C05355=1014.122,185.886,-129.232,167.084,55.090,160.182
C05356=1014.126,186.134,-129.253,167.087,55.079,160.180
C05357=1014.130,186.414,-129.276,167.092,55.066,160.179
C05358=1014.134,186.693,-129.300,167.097,55.052,160.177
C05359=1014.140,186.972,-129.324,167.102,55.039,160.176
C05360=1014.144,187.252,-129.348,167.107,55.025,160.174
C05361=1014.148,187.500,-129.369,167.111,55.014,160.173
C05362=1014.152,187.750,-129.391,167.116,55.002,160.171
C05363=1014.156,187.999,-129.411,167.120,54.990,160.170
C05364=1014.160,188.248,-129.433,167.124,54.979,160.168
C05365=1014.164,188.496,-129.454,167.129,54.967,160.167
C05366=1014.168,188.746,-129.476,167.134,54.955,160.166
C05367=1014.172,188.995,-129.497,167.137,54.943,160.164
C05368=1014.177,189.244,-129.518,167.142,54.931,160.163
C05369=1014.180,189.493,-129.538,167.146,54.920,160.161
C05370=1014.184,189.743,-129.560,167.150,54.908,160.160
C05371=1014.188,189.991,-129.582,167.155,54.896,160.159
C05372=1014.193,190.240,-129.603,167.160,54.885,160.157
C05373=1014.197,190.490,-129.624,167.164,54.873,160.156
C05374=1014.201,190.739,-129.645,167.168,54.861,160.154
C05375=1014.205,190.988,-129.667,167.172,54.849,160.153
C05376=1014.209,191.236,-129.688,167.177,54.837,160.151
C05377=1014.213,191.486,-129.710,167.181,54.826,160.150
C05378=1014.217,191.734,-129.731,167.186,54.814,160.149
C05379=1014.222,191.984,-129.752,167.190,54.802,160.147
C05380=1014.226,192.233,-129.774,167.195,54.790,160.146
C05381=1014.230,192.482,-129.795,167.199,54.778,160.144
C05382=1014.234,192.731,-129.817,167.203,54.767,160.143
C05383=1014.238,192.980,-129.838,167.208,54.755,160.142
C05384=1014.243,193.228,-129.859,167.213,54.743,160.140
C05385=1014.247,193.478,-129.881,167.218,54.731,160.139
C05386=1014.251,193.727,-129.902,167.222,54.719,160.137
C05387=1014.256,193.976,-129.924,167.226,54.707,160.136
C05388=1014.259,194.225,-129.946,167.231,54.696,160.135
C05389=1014.263,194.474,-129.966,167.235,54.684,160.133
C05390=1014.268,194.723,-129.988,167.240,54.672,160.132
C05391=1014.273,194.972,-130.009,167.245,54.660,160.131
C05392=1014.276,195.221,-130.031,167.249,54.648,160.129
C05393=1014.281,195.470,-130.053,167.253,54.637,160.127
C05394=1014.286,195.719,-130.074,167.258,54.625,160.126
C05395=1014.289,195.969,-130.096,167.263,54.613,160.125
C05396=1014.293,196.218,-130.117,167.267,54.601,160.123
C05397=1014.298,196.466,-130.139,167.272,54.589,160.122
C05398=1014.303,196.716,-130.160,167.277,54.577,160.121
C05399=1014.306,196.964,-130.182,167.282,54.565,160.119
C05400=1014.311,197.214,-130.203,167.287,54.554,160.118
C05401=1014.315,197.462,-130.225,167.290,54.542,160.116
C05402=1014.320,197.712,-130.246,167.295,54.530,160.115
C05403=1014.323,197.960,-130.268,167.300,54.518,160.114
C05404=1014.328,198.209,-130.290,167.304,54.507,160.112
C05405=1014.333,198.459,-130.311,167.309,54.495,160.111
C05406=1014.337,198.708,-130.334,167.314,54.482,160.109
C05407=1014.341,198.957,-130.355,167.319,54.471,160.108
C05408=1014.345,199.206,-130.377,167.323,54.459,160.107
C05409=1014.350,199.454,-130.399,167.328,54.447,160.105
C05410=1014.354,199.704,-130.421,167.333,54.436,160.104
C05411=1014.358,199.953,-130.443,167.337,54.424,160.103
C05412=1014.362,200.202,-130.465,167.342,54.413,160.101
C05413=1014.366,200.451,-130.487,167.347,54.401,160.100
C05414=1014.370,200.700,-130.510,167.352,54.389,160.099
C05415=1014.375,200.948,-130.531,167.357,54.378,160.097
C05416=1014.379,201.198,-130.554,167.362,54.366,160.096
C05417=1014.383,201.447,-130.576,167.366,54.354,160.095
C05418=1014.387,201.696,-130.597,167.371,54.342,160.093
C05419=1014.391,201.945,-130.620,167.375,54.331,160.092
C05420=1014.395,202.194,-130.642,167.380,54.319,160.090
C05421=1014.415,203.311,-130.741,167.905,54.401,160.226
C05422=1014.420,203.543,-130.764,167.909,54.392,160.225
C05423=1014.424,203.777,-130.786,167.913,54.381,160.223
C05424=1014.429,204.010,-130.808,167.918,54.371,160.222
C05425=1014.435,204.242,-130.831,167.921,54.361,160.221
C05426=1014.439,204.475,-130.853,167.926,54.351,160.220
C05427=1014.444,204.708,-130.875,167.930,54.341,160.218
C05428=1014.449,204.940,-130.897,167.934,54.331,160.217
C05429=1014.454,205.173,-130.919,167.939,54.322,160.216
C05430=1014.460,205.422,-130.944,167.943,54.311,160.215
C05431=1014.465,205.671,-130.967,167.947,54.301,160.213
C05432=1014.470,205.920,-130.991,167.952,54.290,160.212
C05433=1014.475,206.168,-131.016,167.956,54.280,160.211
C05434=1014.481,206.418,-131.040,167.960,54.269,160.210
C05435=1014.486,206.667,-131.064,167.964,54.258,160.208
C05436=1014.491,206.915,-131.088,167.969,54.248,160.207
C05437=1014.497,207.164,-131.112,167.974,54.237,160.206
C05438=1014.502,207.413,-131.137,167.978,54.227,160.204
C05439=1014.507,207.662,-131.160,167.983,54.217,160.203
C05440=1014.512,207.910,-131.184,167.987,54.206,160.202
C05441=1014.518,208.159,-131.209,167.992,54.196,160.201
C05442=1014.523,208.408,-131.233,167.996,54.185,160.199
C05443=1014.528,208.656,-131.257,168.000,54.175,160.198
C05444=1014.533,208.905,-131.281,168.005,54.165,160.197
C05445=1014.538,209.154,-131.305,168.009,54.154,160.196
C05446=1014.544,209.403,-131.329,168.014,54.144,160.194
C05447=1014.550,209.652,-131.354,168.019,54.134,160.193
C05448=1014.554,209.901,-131.379,168.023,54.124,160.192
C05449=1014.559,210.149,-131.403,168.027,54.113,160.191
C05450=1014.565,210.398,-131.427,168.032,54.103,160.190
C05451=1014.570,210.646,-131.452,168.036,54.093,160.188
C05452=1014.575,210.895,-131.476,168.040,54.083,160.187
C05453=1014.580,211.144,-131.501,168.044,54.073,160.186
C05454=1014.586,211.393,-131.525,168.049,54.063,160.185
C05455=1014.591,211.642,-131.550,168.054,54.053,160.184
C05456=1014.596,211.890,-131.574,168.058,54.042,160.182
C05457=1014.601,212.139,-131.599,168.063,54.032,160.181
C05458=1014.606,212.388,-131.623,168.067,54.022,160.180
C05459=1014.613,212.637,-131.648,168.072,54.012,160.179
C05460=1014.618,212.885,-131.672,168.076,54.002,160.178
C05461=1014.622,213.134,-131.697,168.081,53.992,160.176
C05462=1014.628,213.383,-131.722,168.084,53.982,160.175
C05463=1014.633,213.631,-131.746,168.089,53.972,160.174
C05464=1014.639,213.881,-131.770,168.094,53.962,160.173
C05465=1014.644,214.129,-131.795,168.098,53.952,160.172
C05466=1014.649,214.378,-131.820,168.103,53.942,160.171
C05467=1014.654,214.626,-131.845,168.108,53.932,160.169
C05468=1014.660,214.875,-131.869,168.113,53.922,160.168
C05469=1014.666,215.124,-131.893,168.116,53.913,160.167
C05470=1014.670,215.373,-131.918,168.121,53.902,160.166
C05471=1014.676,215.622,-131.943,168.126,53.892,160.165
C05472=1014.682,215.870,-131.968,168.130,53.883,160.164
C05473=1014.687,216.119,-131.992,168.135,53.872,160.162
C05474=1014.691,216.367,-132.017,168.140,53.863,160.161
C05475=1014.697,216.617,-132.042,168.144,53.853,160.160
C05476=1014.703,216.865,-132.067,168.148,53.843,160.159
C05477=1014.708,217.113,-132.091,168.153,53.833,160.158
C05478=1014.714,217.363,-132.115,168.158,53.823,160.157
C05479=1014.719,217.612,-132.140,168.163,53.814,160.156
C05480=1014.724,217.859,-132.165,168.166,53.803,160.154
C05481=1014.730,218.108,-132.190,168.171,53.794,160.153
C05482=1014.735,218.355,-132.215,168.176,53.784,160.152
C05483=1014.740,218.600,-132.239,168.179,53.775,160.151
C05484=1014.745,218.846,-132.264,168.184,53.765,160.150
C05485=1014.750,219.092,-132.289,168.188,53.756,160.149
C05486=1014.756,219.338,-132.314,168.193,53.746,160.147
C05487=1014.761,219.584,-132.340,168.197,53.737,160.147
C05488=1014.766,219.829,-132.364,168.202,53.728,160.145
C05489=1014.771,220.075,-132.389,168.206,53.718,160.144
C05490=1014.777,220.324,-132.413,168.211,53.709,160.143
C05491=1014.782,220.573,-132.439,168.216,53.699,160.142
C05492=1014.787,220.821,-132.463,168.220,53.690,160.141
C05493=1014.793,221.070,-132.489,168.225,53.680,160.140
C05494=1014.798,221.318,-132.514,168.230,53.670,160.139
C05495=1014.803,221.568,-132.539,168.234,53.661,160.138
C05496=1014.809,221.816,-132.564,168.238,53.651,160.137
C05497=1014.814,222.065,-132.590,168.243,53.641,160.136
C05498=1014.820,222.313,-132.615,168.247,53.632,160.134
C05499=1014.825,222.562,-132.640,168.252,53.622,160.133
C05500=1014.831,222.811,-132.665,168.257,53.614,160.132
C05501=1014.835,223.059,-132.690,168.261,53.604,160.131
C05502=1014.842,223.308,-132.716,168.266,53.594,160.130
C05503=1014.846,223.557,-132.740,168.270,53.585,160.129
C05504=1014.852,223.806,-132.766,168.275,53.575,160.128
C05505=1014.857,224.054,-132.791,168.279,53.566,160.127
C05506=1014.862,224.303,-132.817,168.285,53.557,160.126
C05507=1014.868,224.551,-132.842,168.288,53.548,160.125
C05508=1014.873,224.800,-132.868,168.293,53.538,160.124
C05509=1014.880,225.049,-132.893,168.298,53.528,160.123
C05510=1014.884,225.298,-132.918,168.303,53.520,160.122
C05511=1014.890,225.547,-132.943,168.308,53.510,160.121
C05512=1014.895,225.795,-132.969,168.312,53.501,160.120
C05513=1014.902,226.044,-132.994,168.317,53.492,160.119
C05514=1014.906,226.292,-133.020,168.321,53.483,160.118
C05515=1014.912,226.541,-133.045,168.326,53.473,160.117
C05516=1014.916,226.790,-133.070,168.330,53.464,160.116
C05517=1014.922,227.039,-133.096,168.335,53.455,160.115
C05518=1014.928,227.287,-133.122,168.340,53.446,160.114
C05519=1014.933,227.536,-133.147,168.343,53.437,160.112
C05520=1014.938,227.785,-133.173,168.349,53.428,160.112
C05521=1014.943,228.033,-133.199,168.353,53.419,160.110
C05522=1014.949,228.282,-133.224,168.358,53.410,160.110
C05523=1014.955,228.531,-133.250,168.362,53.400,160.108
C05524=1014.960,228.779,-133.275,168.368,53.392,160.108
C05525=1014.965,229.028,-133.301,168.372,53.382,160.106
C05526=1014.970,229.276,-133.327,168.376,53.374,160.105
C05527=1014.977,229.524,-133.353,168.381,53.365,160.105
C05528=1014.982,229.773,-133.379,168.385,53.355,160.103
C05529=1014.987,230.021,-133.405,168.391,53.347,160.103
C05530=1014.992,230.270,-133.430,168.395,53.338,160.102
C05531=1014.998,230.519,-133.456,168.399,53.329,160.101
C05532=1015.003,230.768,-133.482,168.405,53.320,160.100
C05533=1015.009,231.016,-133.509,168.409,53.311,160.099
C05534=1015.014,231.265,-133.535,168.413,53.303,160.098
C05535=1015.019,231.513,-133.560,168.418,53.293,160.097
C05536=1015.024,231.762,-133.586,168.423,53.284,160.096
C05537=1015.030,232.011,-133.612,168.427,53.276,160.095
C05538=1015.035,232.259,-133.638,168.432,53.267,160.094
C05539=1015.040,232.508,-133.664,168.437,53.258,160.093
C05540=1015.046,232.757,-133.690,168.441,53.249,160.092
C05541=1015.051,233.004,-133.716,168.445,53.241,160.091
C05542=1015.057,233.246,-133.742,168.450,53.232,160.090
C05543=1015.062,233.488,-133.767,168.454,53.224,160.089
C05544=1015.068,233.730,-133.792,168.460,53.215,160.088
C05545=1015.072,233.972,-133.818,168.465,53.207,160.088
C05546=1015.078,234.213,-133.843,168.469,53.198,160.087
C05547=1015.083,234.455,-133.868,168.474,53.190,160.086
C05548=1015.089,234.697,-133.893,168.478,53.181,160.085
C05549=1015.094,234.938,-133.918,168.483,53.173,160.084
C05550=1015.100,235.187,-133.945,168.487,53.164,160.083
C05551=1015.105,235.436,-133.971,168.491,53.156,160.082
C05552=1015.111,235.684,-133.997,168.497,53.147,160.081
C05553=1015.116,235.933,-134.023,168.501,53.138,160.080
C05554=1015.121,236.181,-134.049,168.506,53.130,160.079
C05555=1015.127,236.430,-134.075,168.510,53.121,160.078
C05556=1015.132,236.679,-134.101,168.515,53.113,160.077
C05557=1015.138,236.927,-134.128,168.520,53.104,160.076
C05558=1015.144,237.176,-134.154,168.525,53.095,160.076
C05559=1015.149,237.424,-134.181,168.530,53.087,160.075
C05560=1015.154,237.673,-134.206,168.534,53.079,160.074
C05561=1015.159,237.921,-134.233,168.538,53.070,160.073
C05562=1015.165,238.170,-134.260,168.544,53.061,160.072
C05563=1015.171,238.419,-134.286,168.548,53.053,160.071
C05564=1015.176,238.667,-134.313,168.553,53.044,160.070
C05565=1015.182,238.915,-134.339,168.558,53.037,160.070
C05566=1015.187,239.164,-134.365,168.562,53.028,160.069
C05567=1015.193,239.412,-134.392,168.567,53.020,160.068
C05568=1015.198,239.661,-134.419,168.572,53.012,160.067
C05569=1015.204,239.909,-134.445,168.576,53.003,160.066
C05570=1015.209,240.158,-134.471,168.582,52.994,160.065
C05571=1015.214,240.407,-134.499,168.587,52.987,160.064
C05572=1015.220,240.655,-134.525,168.591,52.978,160.064
C05573=1015.226,240.903,-134.552,168.596,52.970,160.063
C05574=1015.230,241.153,-134.578,168.600,52.962,160.062
C05575=1015.236,241.401,-134.605,168.605,52.953,160.061
C05576=1015.242,241.649,-134.632,168.610,52.946,160.060
C05577=1015.248,241.898,-134.658,168.614,52.937,160.059
C05578=1015.253,242.146,-134.686,168.619,52.929,160.059
C05579=1015.258,242.394,-134.712,168.624,52.921,160.058
C05580=1015.264,242.642,-134.739,168.629,52.913,160.057
C05581=1015.269,242.891,-134.766,168.633,52.905,160.056
C05582=1015.275,243.139,-134.792,168.638,52.897,160.055
C05583=1015.280,243.388,-134.820,168.643,52.888,160.054
C05584=1015.285,243.636,-134.846,168.648,52.880,160.054
C05585=1015.290,243.885,-134.874,168.653,52.873,160.053
C05586=1015.295,244.134,-134.901,168.657,52.864,160.052
C05587=1015.301,244.382,-134.927,168.662,52.856,160.051
C05588=1015.306,244.631,-134.955,168.667,52.849,160.051
C05589=1015.312,244.879,-134.981,168.672,52.841,160.050
C05590=1015.317,245.127,-135.009,168.676,52.832,160.049
C05591=1015.322,245.376,-135.037,168.681,52.825,160.048
C05592=1015.328,245.624,-135.063,168.686,52.817,160.047
C05593=1015.333,245.873,-135.090,168.691,52.809,160.047
C05594=1015.339,246.121,-135.117,168.696,52.801,160.046
C05595=1015.344,246.370,-135.144,168.701,52.793,160.045
C05596=1015.350,246.619,-135.173,168.705,52.785,160.044
C05597=1015.356,246.867,-135.199,168.710,52.778,160.044
C05598=1015.361,247.116,-135.227,168.715,52.770,160.043
C05599=1015.367,247.364,-135.253,168.719,52.761,160.042
C05600=1015.372,247.612,-135.281,168.724,52.754,160.041
C05601=1015.378,247.861,-135.308,168.729,52.746,160.040
C05602=1015.383,248.098,-135.334,168.734,52.738,160.040
C05603=1015.388,248.338,-135.360,168.739,52.731,160.039
C05604=1015.393,248.576,-135.386,168.743,52.724,160.038
C05605=1015.398,248.814,-135.412,168.747,52.716,160.038
C05606=1015.404,249.052,-135.439,168.752,52.708,160.037
C05607=1015.409,249.290,-135.465,168.756,52.701,160.036
C05608=1015.414,249.529,-135.492,168.762,52.694,160.036
C05609=1015.419,249.768,-135.517,168.767,52.686,160.035
C05610=1015.425,250.015,-135.545,168.771,52.679,160.034
C05611=1015.430,250.264,-135.572,168.776,52.671,160.033
C05612=1015.437,250.512,-135.600,168.781,52.663,160.033
C05613=1015.442,250.761,-135.627,168.786,52.656,160.032
C05614=1015.447,251.010,-135.654,168.791,52.648,160.031
C05615=1015.453,251.257,-135.681,168.796,52.640,160.030
C05616=1015.458,251.506,-135.709,168.801,52.632,160.030
C05617=1015.465,251.755,-135.736,168.806,52.625,160.029
C05618=1015.470,252.003,-135.764,168.810,52.617,160.028
C05619=1015.475,252.251,-135.792,168.815,52.610,160.027
C05620=1015.481,252.500,-135.818,168.820,52.602,160.027
C05621=1015.487,252.748,-135.847,168.825,52.595,160.026
C05622=1015.493,252.997,-135.873,168.830,52.587,160.026
C05623=1015.498,253.245,-135.901,168.835,52.579,160.025
C05624=1015.504,253.494,-135.929,168.840,52.572,160.024
C05625=1015.510,253.742,-135.956,168.844,52.564,160.023
C05626=1015.515,253.991,-135.983,168.849,52.556,160.023
C05627=1015.521,254.239,-136.012,168.854,52.549,160.022
C05628=1015.527,254.488,-136.038,168.859,52.542,160.021
C05629=1015.532,254.736,-136.066,168.864,52.534,160.021
C05630=1015.539,254.984,-136.094,168.869,52.526,160.020
C05631=1015.544,255.233,-136.121,168.874,52.519,160.019
C05632=1015.549,255.481,-136.149,168.879,52.512,160.019
C05633=1015.555,255.730,-136.176,168.884,52.504,160.018
C05634=1015.561,255.978,-136.204,168.889,52.496,160.017
C05635=1015.567,256.226,-136.232,168.894,52.489,160.017
C05636=1015.572,256.475,-136.259,168.899,52.482,160.016
C05637=1015.578,256.723,-136.287,168.903,52.474,160.015
C05638=1015.584,256.972,-136.315,168.909,52.467,160.015
C05639=1015.590,257.220,-136.343,168.914,52.460,160.014
C05640=1015.595,257.469,-136.370,168.919,52.452,160.013
C05641=1015.601,257.717,-136.398,168.924,52.445,160.013
C05642=1015.607,257.965,-136.426,168.929,52.437,160.012
C05643=1015.613,258.213,-136.454,168.933,52.430,160.011
C05644=1015.618,258.462,-136.481,168.939,52.423,160.011
C05645=1015.624,258.711,-136.509,168.944,52.415,160.010
C05646=1015.631,258.958,-136.536,168.949,52.408,160.009
C05647=1015.636,259.207,-136.565,168.954,52.400,160.009
C05648=1015.643,259.455,-136.592,168.959,52.394,160.008
C05649=1015.648,259.703,-136.620,168.964,52.386,160.007
C05650=1015.654,259.952,-136.648,168.969,52.379,160.007
C05651=1015.659,260.200,-136.676,168.974,52.372,160.006
C05652=1015.665,260.449,-136.705,168.979,52.365,160.006
C05653=1015.670,260.697,-136.733,168.984,52.358,160.005
C05654=1015.676,260.945,-136.761,168.988,52.351,160.004
C05655=1015.682,261.193,-136.789,168.994,52.343,160.004
C05656=1015.688,261.442,-136.818,168.999,52.336,160.003
C05657=1015.693,261.690,-136.846,169.003,52.330,160.003
C05658=1015.699,261.938,-136.874,169.009,52.323,160.002
C05659=1015.704,262.187,-136.903,169.014,52.315,160.001
C05660=1015.710,262.435,-136.931,169.018,52.308,160.001
C05661=1015.715,262.683,-136.959,169.024,52.301,160.000
C05662=1015.721,262.921,-136.986,169.028,52.295,160.000
C05663=1015.727,263.158,-137.014,169.034,52.288,159.999
C05664=1015.732,263.396,-137.041,169.038,52.281,159.999
C05665=1015.737,263.633,-137.068,169.043,52.274,159.998
C05666=1015.743,263.870,-137.095,169.049,52.268,159.998
C05667=1015.748,264.108,-137.122,169.053,52.261,159.997
C05668=1015.754,264.345,-137.149,169.058,52.255,159.997
C05669=1015.760,264.582,-137.177,169.063,52.248,159.996
C05670=1015.765,264.830,-137.205,169.067,52.241,159.995
C05671=1015.771,265.079,-137.233,169.073,52.234,159.995
C05672=1015.777,265.326,-137.262,169.077,52.228,159.994
C05673=1015.783,265.575,-137.290,169.083,52.221,159.994
C05674=1015.788,265.824,-137.320,169.088,52.214,159.993
C05675=1015.794,266.072,-137.348,169.093,52.207,159.993
C05676=1015.799,266.320,-137.376,169.098,52.200,159.992
C05677=1015.806,266.569,-137.405,169.103,52.193,159.992
C05678=1015.811,266.817,-137.433,169.108,52.186,159.991
C05679=1015.817,267.065,-137.463,169.114,52.179,159.991
C05680=1015.823,267.314,-137.491,169.119,52.173,159.990
C05681=1015.828,267.561,-137.520,169.124,52.166,159.990
C05682=1015.834,267.810,-137.548,169.129,52.160,159.989
C05683=1015.840,268.058,-137.577,169.134,52.153,159.989
C05684=1015.846,268.307,-137.607,169.140,52.146,159.988
C05685=1015.851,268.555,-137.635,169.144,52.139,159.987
C05686=1015.857,268.803,-137.664,169.150,52.132,159.987
C05687=1015.863,269.052,-137.692,169.154,52.126,159.987
C05688=1015.868,269.299,-137.721,169.160,52.119,159.986
C05689=1015.875,269.547,-137.750,169.164,52.113,159.985
C05690=1015.880,269.796,-137.780,169.170,52.106,159.985
C05691=1015.886,270.045,-137.808,169.175,52.100,159.985
C05692=1015.892,270.292,-137.837,169.180,52.093,159.984
C05693=1015.897,270.540,-137.867,169.185,52.087,159.984
C05694=1015.903,270.789,-137.896,169.191,52.080,159.983
C05695=1015.909,271.037,-137.924,169.196,52.073,159.983
C05696=1015.915,271.286,-137.954,169.201,52.067,159.982
C05697=1015.921,271.533,-137.982,169.207,52.060,159.982
C05698=1015.926,271.782,-138.012,169.211,52.054,159.981
C05699=1015.932,272.030,-138.041,169.217,52.047,159.981
C05700=1015.939,272.278,-138.070,169.222,52.041,159.980
C05701=1015.944,272.527,-138.099,169.228,52.034,159.980
C05702=1015.949,272.774,-138.128,169.232,52.028,159.979
C05703=1015.955,273.023,-138.157,169.238,52.021,159.979
C05704=1015.961,273.271,-138.186,169.242,52.015,159.978
C05705=1015.967,273.519,-138.216,169.248,52.009,159.978
C05706=1015.973,273.768,-138.245,169.253,52.002,159.978
C05707=1015.978,274.016,-138.275,169.259,51.996,159.977
C05708=1015.985,274.264,-138.304,169.264,51.990,159.977
C05709=1015.990,274.513,-138.333,169.269,51.983,159.976
C05710=1015.996,274.761,-138.362,169.274,51.977,159.976
C05711=1016.001,275.008,-138.391,169.280,51.970,159.975
C05712=1016.008,275.257,-138.421,169.285,51.964,159.975
C05713=1016.013,275.505,-138.450,169.291,51.958,159.975
C05714=1016.020,275.753,-138.480,169.295,51.951,159.974
C05715=1016.026,276.001,-138.509,169.301,51.945,159.974
C05716=1016.031,276.249,-138.539,169.306,51.939,159.974
C05717=1016.037,276.498,-138.568,169.310,51.933,159.973
C05718=1016.043,276.746,-138.597,169.316,51.926,159.973
C05719=1016.049,276.994,-138.628,169.321,51.920,159.972
C05720=1016.054,277.242,-138.657,169.327,51.914,159.972
C05721=1016.060,277.490,-138.687,169.332,51.908,159.972
C05722=1016.066,277.729,-138.715,169.337,51.902,159.971
C05723=1016.071,277.970,-138.744,169.342,51.896,159.971
C05724=1016.077,278.209,-138.773,169.348,51.890,159.970
C05725=1016.082,278.448,-138.802,169.353,51.884,159.970
C05726=1016.089,278.688,-138.830,169.358,51.878,159.970
C05727=1016.094,278.927,-138.859,169.363,51.872,159.969
C05728=1016.100,279.167,-138.888,169.368,51.867,159.969
C05729=1016.105,279.406,-138.916,169.373,51.861,159.968
C05730=1016.111,279.655,-138.946,169.379,51.854,159.968
C05731=1016.117,279.903,-138.976,169.383,51.849,159.968
C05732=1016.123,280.151,-139.006,169.389,51.842,159.967
C05733=1016.129,280.399,-139.036,169.394,51.836,159.967
C05734=1016.134,280.647,-139.066,169.400,51.830,159.967
C05735=1016.141,280.895,-139.096,169.405,51.824,159.966
C05736=1016.147,281.144,-139.125,169.410,51.818,159.966
C05737=1016.153,281.391,-139.156,169.416,51.812,159.966
C05738=1016.158,281.640,-139.185,169.421,51.806,159.965
C05739=1016.165,281.887,-139.215,169.427,51.800,159.965
C05740=1016.170,282.136,-139.245,169.432,51.794,159.965
C05741=1016.176,282.384,-139.275,169.437,51.788,159.964
C05742=1016.182,282.633,-139.305,169.443,51.783,159.964
C05743=1016.189,282.880,-139.335,169.448,51.777,159.964
C05744=1016.195,283.128,-139.365,169.454,51.771,159.963
C05745=1016.200,283.377,-139.395,169.459,51.765,159.963
C05746=1016.206,283.624,-139.425,169.465,51.758,159.963
C05747=1016.212,283.872,-139.455,169.470,51.753,159.962
C05748=1016.219,284.121,-139.485,169.475,51.747,159.962
C05749=1016.224,284.369,-139.515,169.481,51.741,159.962
C05750=1016.230,284.617,-139.546,169.486,51.735,159.961
C05751=1016.236,284.865,-139.576,169.492,51.729,159.961
C05752=1016.242,285.114,-139.606,169.498,51.724,159.961
C05753=1016.248,285.361,-139.636,169.503,51.718,159.961
C05754=1016.254,285.609,-139.667,169.508,51.712,159.960
C05755=1016.260,285.857,-139.696,169.514,51.707,159.960
C05756=1016.267,286.105,-139.727,169.519,51.701,159.960
C05757=1016.273,286.353,-139.757,169.525,51.695,159.960
C05758=1016.278,286.601,-139.788,169.530,51.689,159.959
C05759=1016.284,286.849,-139.818,169.535,51.683,159.959
C05760=1016.291,287.097,-139.849,169.541,51.678,159.959
C05761=1016.296,287.345,-139.879,169.546,51.672,159.958
C05762=1016.302,287.593,-139.910,169.552,51.667,159.958
C05763=1016.309,287.841,-139.940,169.558,51.661,159.958
C05764=1016.315,288.089,-139.971,169.563,51.655,159.958
C05765=1016.320,288.337,-140.001,169.568,51.650,159.957
C05766=1016.326,288.586,-140.032,169.574,51.644,159.957
C05767=1016.332,288.834,-140.063,169.579,51.638,159.957
C05768=1016.338,289.082,-140.093,169.586,51.633,159.957
C05769=1016.344,289.330,-140.124,169.591,51.627,159.957
C05770=1016.350,289.578,-140.154,169.596,51.622,159.956
C05771=1016.356,289.825,-140.185,169.602,51.616,159.956
C05772=1016.362,290.074,-140.216,169.607,51.610,159.956
C05773=1016.368,290.321,-140.246,169.613,51.605,159.955
C05774=1016.375,290.570,-140.277,169.619,51.599,159.955
C05775=1016.380,290.818,-140.307,169.624,51.594,159.955
C05776=1016.387,291.065,-140.338,169.630,51.588,159.955
C05777=1016.393,291.314,-140.369,169.636,51.583,159.955
C05778=1016.398,291.562,-140.400,169.641,51.578,159.955
C05779=1016.405,291.810,-140.431,169.646,51.572,159.954
C05780=1016.411,292.057,-140.462,169.653,51.566,159.954
C05781=1016.417,292.306,-140.492,169.658,51.561,159.954
C05782=1016.423,292.551,-140.523,169.663,51.556,159.954
C05783=1016.429,292.797,-140.554,169.669,51.551,159.953
C05784=1016.435,293.043,-140.584,169.675,51.545,159.953
C05785=1016.441,293.289,-140.616,169.681,51.540,159.953
C05786=1016.446,293.534,-140.647,169.686,51.535,159.953
C05787=1016.453,293.779,-140.678,169.691,51.530,159.953
C05788=1016.458,294.026,-140.708,169.697,51.524,159.953
C05789=1016.464,294.272,-140.740,169.702,51.519,159.952
C05790=1016.470,294.519,-140.771,169.708,51.514,159.952
C05791=1016.476,294.767,-140.803,169.714,51.509,159.952
C05792=1016.482,295.015,-140.833,169.719,51.503,159.952
C05793=1016.488,295.263,-140.865,169.725,51.498,159.952
C05794=1016.493,295.511,-140.897,169.731,51.493,159.952
C05795=1016.500,295.759,-140.928,169.736,51.488,159.951
C05796=1016.505,296.007,-140.959,169.742,51.482,159.951
C05797=1016.512,296.255,-140.991,169.748,51.478,159.951
C05798=1016.518,296.503,-141.023,169.754,51.472,159.951
C05799=1016.524,296.750,-141.054,169.759,51.467,159.951
C05800=1016.530,296.999,-141.085,169.765,51.462,159.951
C05801=1016.536,297.246,-141.116,169.770,51.457,159.951
C05802=1016.542,297.494,-141.148,169.777,51.452,159.951
C05803=1016.549,297.742,-141.180,169.782,51.447,159.951
C05804=1016.554,297.990,-141.211,169.788,51.442,159.950
C05805=1016.561,298.238,-141.243,169.793,51.437,159.950
C05806=1016.567,298.486,-141.275,169.799,51.431,159.950
C05807=1016.572,298.733,-141.306,169.805,51.427,159.950
C05808=1016.579,298.981,-141.338,169.811,51.421,159.950
C05809=1016.585,299.229,-141.370,169.816,51.416,159.950
C05810=1016.591,299.477,-141.401,169.823,51.411,159.950
C05811=1016.597,299.725,-141.433,169.828,51.406,159.950
C05812=1016.604,299.973,-141.464,169.834,51.401,159.949
C05813=1016.610,300.221,-141.496,169.840,51.396,159.950
C05814=1016.616,300.468,-141.528,169.846,51.391,159.949
C05815=1016.622,300.716,-141.560,169.852,51.387,159.949
C05816=1016.628,300.964,-141.591,169.857,51.381,159.949
C05817=1016.634,301.212,-141.623,169.863,51.376,159.949
C05818=1016.640,301.460,-141.655,169.869,51.371,159.949
C05819=1016.647,301.708,-141.686,169.875,51.366,159.949
C05820=1016.653,301.956,-141.718,169.880,51.362,159.949
C05821=1016.659,302.204,-141.750,169.887,51.356,159.949
C05822=1016.665,302.452,-141.782,169.893,51.352,159.949
C05823=1016.672,302.699,-141.813,169.898,51.347,159.949
C05824=1016.678,302.947,-141.845,169.905,51.342,159.949
C05825=1016.684,303.195,-141.877,169.910,51.337,159.949
C05826=1016.690,303.443,-141.909,169.916,51.332,159.949
C05827=1016.697,303.690,-141.941,169.921,51.327,159.948
C05828=1016.703,303.939,-141.973,169.928,51.322,159.949
C05829=1016.709,304.187,-142.005,169.934,51.318,159.949
C05830=1016.716,304.435,-142.037,169.939,51.313,159.948
C05831=1016.722,304.682,-142.069,169.946,51.308,159.948
C05832=1016.729,304.929,-142.100,169.952,51.303,159.948
C05833=1016.735,305.178,-142.132,169.957,51.298,159.948
C05834=1016.742,305.425,-142.165,169.963,51.294,159.948
C05835=1016.748,305.673,-142.197,169.970,51.288,159.948
C05836=1016.755,305.920,-142.229,169.975,51.284,159.948
C05837=1016.761,306.169,-142.261,169.981,51.279,159.948
C05838=1016.767,306.417,-142.293,169.988,51.274,159.948
C05839=1016.774,306.664,-142.325,169.993,51.269,159.948
C05840=1016.780,306.912,-142.357,169.999,51.265,159.948
C05841=1016.787,307.160,-142.389,170.005,51.260,159.948
C05842=1016.793,307.422,-142.423,170.011,51.255,159.948
C05843=1016.800,307.682,-142.457,170.018,51.250,159.948
C05844=1016.807,307.944,-142.491,170.025,51.245,159.948
C05845=1016.814,308.206,-142.525,170.030,51.240,159.948
C05846=1016.821,308.453,-142.557,170.037,51.235,159.948
C05847=1016.827,308.701,-142.590,170.043,51.231,159.948
C05848=1016.834,308.949,-142.621,170.049,51.226,159.948
C05849=1016.840,309.196,-142.654,170.056,51.221,159.948
C05850=1016.847,309.444,-142.685,170.061,51.217,159.948
C05851=1016.853,309.692,-142.718,170.067,51.212,159.948
C05852=1016.859,309.940,-142.752,170.073,51.208,159.948
C05853=1016.865,310.187,-142.784,170.080,51.203,159.948
C05854=1016.871,310.435,-142.817,170.086,51.199,159.948
C05855=1016.878,310.683,-142.850,170.092,51.194,159.948
C05856=1016.884,310.930,-142.882,170.098,51.190,159.949
C05857=1016.890,311.179,-142.916,170.104,51.186,159.949
C05858=1016.896,311.426,-142.949,170.109,51.182,159.949
C05859=1016.903,311.674,-142.982,170.116,51.177,159.949
C05860=1016.909,311.921,-143.015,170.122,51.173,159.949
C05861=1016.916,312.169,-143.048,170.128,51.168,159.949
C05862=1016.921,312.416,-143.081,170.134,51.164,159.949
C05863=1016.928,312.664,-143.114,170.140,51.159,159.949
C05864=1016.934,312.912,-143.147,170.147,51.155,159.949
C05865=1016.941,313.160,-143.180,170.153,51.151,159.949
C05866=1016.947,313.408,-143.213,170.159,51.147,159.950
C05867=1016.953,313.655,-143.247,170.165,51.143,159.950
C05868=1016.959,313.902,-143.279,170.172,51.138,159.950
C05869=1016.966,314.151,-143.312,170.178,51.134,159.950
C05870=1016.972,314.398,-143.345,170.184,51.130,159.950
C05871=1016.979,314.645,-143.379,170.190,51.126,159.950
C05872=1016.984,314.893,-143.412,170.196,51.121,159.950
C05873=1016.991,315.141,-143.445,170.203,51.116,159.950
C05874=1016.998,315.388,-143.479,170.209,51.113,159.950
C05875=1017.004,315.636,-143.511,170.215,51.108,159.950
C05876=1017.011,315.884,-143.544,170.221,51.104,159.951
C05877=1017.017,316.132,-143.578,170.228,51.100,159.951
C05878=1017.023,316.379,-143.611,170.234,51.096,159.951
C05879=1017.031,316.627,-143.645,170.240,51.092,159.951
C05880=1017.037,316.874,-143.678,170.246,51.088,159.951
C05881=1017.043,317.123,-143.711,170.253,51.083,159.952
C05882=1017.050,317.370,-143.745,170.259,51.079,159.952
C05883=1017.056,317.618,-143.778,170.265,51.075,159.952
C05884=1017.063,317.865,-143.812,170.271,51.071,159.952
C05885=1017.069,318.113,-143.844,170.278,51.067,159.952
C05886=1017.076,318.361,-143.879,170.284,51.063,159.952
C05887=1017.082,318.609,-143.911,170.290,51.058,159.952
C05888=1017.089,318.856,-143.945,170.297,51.054,159.953
C05889=1017.096,319.103,-143.979,170.304,51.050,159.953
C05890=1017.102,319.352,-144.012,170.310,51.047,159.953
C05891=1017.109,319.599,-144.046,170.316,51.042,159.953
C05892=1017.116,319.846,-144.080,170.323,51.038,159.953
C05893=1017.122,320.094,-144.112,170.329,51.034,159.954
C05894=1017.129,320.342,-144.146,170.335,51.030,159.954
C05895=1017.135,320.589,-144.180,170.341,51.026,159.954
C05896=1017.142,320.837,-144.213,170.348,51.022,159.954
C05897=1017.149,321.085,-144.247,170.355,51.018,159.954
C05898=1017.156,321.332,-144.281,170.361,51.014,159.954
C05899=1017.162,321.580,-144.315,170.368,51.010,159.955
C05900=1017.169,321.827,-144.348,170.374,51.006,159.955
C05901=1017.176,322.075,-144.382,170.380,51.002,159.955
C05902=1017.183,322.342,-144.419,170.387,50.998,159.955
C05903=1017.190,322.608,-144.455,170.394,50.994,159.956
C05904=1017.198,322.875,-144.491,170.402,50.989,159.956
C05905=1017.205,323.142,-144.527,170.409,50.985,159.956
C05906=1017.212,323.389,-144.561,170.415,50.981,159.956
C05907=1017.219,323.638,-144.594,170.421,50.978,159.957
C05908=1017.225,323.885,-144.628,170.429,50.974,159.957
C05909=1017.232,324.133,-144.662,170.435,50.970,159.957
C05910=1017.239,324.380,-144.696,170.441,50.966,159.957
C05911=1017.246,324.628,-144.730,170.448,50.962,159.958
C05912=1017.253,324.876,-144.764,170.454,50.958,159.958
C05913=1017.260,325.123,-144.798,170.461,50.954,159.958
C05914=1017.267,325.371,-144.832,170.468,50.950,159.958
C05915=1017.274,325.618,-144.865,170.474,50.946,159.959
C05916=1017.281,325.866,-144.901,170.480,50.943,159.959
C05917=1017.288,326.113,-144.934,170.488,50.939,159.959
C05918=1017.295,326.360,-144.968,170.494,50.935,159.960
C05919=1017.301,326.608,-145.002,170.500,50.931,159.960
C05920=1017.308,326.856,-145.037,170.508,50.927,159.960
C05921=1017.315,327.103,-145.071,170.514,50.924,159.960
C05922=1017.321,327.351,-145.106,170.520,50.920,159.961
C05923=1017.328,327.599,-145.141,170.528,50.917,159.961
C05924=1017.335,327.846,-145.174,170.534,50.913,159.961
C05925=1017.342,328.093,-145.209,170.540,50.909,159.962
C05926=1017.348,328.341,-145.244,170.547,50.906,159.962
C05927=1017.356,328.588,-145.278,170.554,50.902,159.962
C05928=1017.362,328.836,-145.313,170.561,50.899,159.963
C05929=1017.369,329.083,-145.348,170.567,50.895,159.963
C05930=1017.375,329.331,-145.382,170.575,50.892,159.963
C05931=1017.383,329.578,-145.417,170.581,50.888,159.964
C05932=1017.389,329.826,-145.451,170.588,50.885,159.964
C05933=1017.396,330.074,-145.486,170.595,50.881,159.964
C05934=1017.403,330.321,-145.521,170.601,50.878,159.965
C05935=1017.410,330.569,-145.555,170.608,50.874,159.965
C05936=1017.417,330.816,-145.591,170.615,50.870,159.965
C05937=1017.424,331.063,-145.625,170.622,50.867,159.966
C05938=1017.431,331.311,-145.659,170.629,50.864,159.966
C05939=1017.437,331.559,-145.695,170.636,50.860,159.967
C05940=1017.444,331.806,-145.730,170.642,50.857,159.967
C05941=1017.451,332.054,-145.764,170.649,50.854,159.967
C05942=1017.458,332.301,-145.799,170.656,50.850,159.968
C05943=1017.465,332.548,-145.834,170.663,50.846,159.968
C05944=1017.472,332.796,-145.869,170.669,50.843,159.969
C05945=1017.478,333.043,-145.904,170.677,50.840,159.969
C05946=1017.487,333.291,-145.939,170.684,50.837,159.969
C05947=1017.493,333.538,-145.974,170.690,50.833,159.970
C05948=1017.500,333.786,-146.009,170.698,50.829,159.970
C05949=1017.507,334.033,-146.044,170.704,50.826,159.971
C05950=1017.514,334.280,-146.080,170.711,50.823,159.971
C05951=1017.520,334.528,-146.115,170.718,50.820,159.971
C05952=1017.527,334.775,-146.150,170.725,50.817,159.972
C05953=1017.535,335.023,-146.185,170.732,50.813,159.972
C05954=1017.541,335.270,-146.220,170.739,50.810,159.973
C05955=1017.548,335.517,-146.256,170.746,50.807,159.973
C05956=1017.555,335.765,-146.291,170.752,50.804,159.974
C05957=1017.563,336.013,-146.327,170.760,50.800,159.974
C05958=1017.569,336.260,-146.362,170.767,50.797,159.975
C05959=1017.576,336.507,-146.397,170.773,50.794,159.975
C05960=1017.583,336.754,-146.433,170.781,50.790,159.975
C05961=1017.590,337.002,-146.469,170.788,50.787,159.976
C05962=1017.598,337.265,-146.506,170.796,50.785,159.977
C05963=1017.606,337.527,-146.543,170.803,50.781,159.977
C05964=1017.613,337.790,-146.581,170.811,50.778,159.978
C05965=1017.620,338.052,-146.619,170.818,50.774,159.978
C05966=1017.627,338.300,-146.654,170.825,50.771,159.978
C05967=1017.635,338.547,-146.690,170.832,50.768,159.979
C05968=1017.642,338.795,-146.726,170.840,50.765,159.980
C05969=1017.649,339.042,-146.762,170.846,50.762,159.980
C05970=1017.656,339.289,-146.797,170.854,50.758,159.981
C05971=1017.663,339.536,-146.833,170.861,50.756,159.981
C05972=1017.671,339.783,-146.869,170.868,50.753,159.982
C05973=1017.678,340.031,-146.904,170.875,50.749,159.982
C05974=1017.684,340.278,-146.941,170.882,50.747,159.983
C05975=1017.691,340.526,-146.976,170.890,50.743,159.983
C05976=1017.699,340.773,-147.012,170.897,50.741,159.984
C05977=1017.706,341.020,-147.048,170.903,50.738,159.984
C05978=1017.713,341.267,-147.084,170.911,50.735,159.985
C05979=1017.719,341.515,-147.120,170.918,50.732,159.985
C05980=1017.727,341.762,-147.156,170.926,50.729,159.986
C05981=1017.734,342.009,-147.192,170.933,50.726,159.986
C05982=1017.742,342.256,-147.228,170.941,50.723,159.987
C05983=1017.748,342.504,-147.265,170.947,50.720,159.988
C05984=1017.756,342.751,-147.301,170.954,50.717,159.988
C05985=1017.764,342.998,-147.337,170.962,50.715,159.989
C05986=1017.771,343.245,-147.373,170.969,50.711,159.989
C05987=1017.778,343.493,-147.410,170.977,50.709,159.990
C05988=1017.785,343.740,-147.446,170.984,50.706,159.991
C05989=1017.792,343.987,-147.482,170.992,50.703,159.991
C05990=1017.799,344.235,-147.519,170.999,50.700,159.992
C05991=1017.806,344.482,-147.555,171.007,50.697,159.992
C05992=1017.814,344.729,-147.591,171.014,50.695,159.993
C05993=1017.821,344.977,-147.628,171.021,50.692,159.994
C05994=1017.828,345.224,-147.663,171.028,50.689,159.994
C05995=1017.836,345.471,-147.700,171.035,50.686,159.995
C05996=1017.843,345.719,-147.736,171.043,50.684,159.995
C05997=1017.850,345.966,-147.773,171.050,50.681,159.996
C05998=1017.858,346.212,-147.809,171.058,50.678,159.997
C05999=1017.865,346.460,-147.845,171.065,50.676,159.997
C06000=1017.872,346.708,-147.882,171.073,50.673,159.998
C06001=1017.880,346.954,-147.919,171.080,50.671,159.999
C06002=1017.887,347.201,-147.956,171.088,50.668,159.999
C06003=1017.894,347.449,-147.992,171.095,50.665,160.000
C06004=1017.902,347.696,-148.029,171.103,50.662,160.001
C06005=1017.909,347.943,-148.066,171.110,50.660,160.001
C06006=1017.916,348.191,-148.103,171.118,50.657,160.002
C06007=1017.924,348.438,-148.139,171.125,50.655,160.003
C06008=1017.931,348.684,-148.176,171.133,50.652,160.003
C06009=1017.938,348.932,-148.213,171.140,50.649,160.004
C06010=1017.946,349.179,-148.250,171.149,50.647,160.005
C06011=1017.953,349.426,-148.288,171.156,50.645,160.005
C06012=1017.961,349.674,-148.324,171.164,50.642,160.006
C06013=1017.968,349.921,-148.361,171.172,50.639,160.007
C06014=1017.976,350.168,-148.398,171.179,50.637,160.008
C06015=1017.983,350.415,-148.435,171.187,50.634,160.008
C06016=1017.991,350.662,-148.472,171.194,50.632,160.009
C06017=1017.998,350.909,-148.510,171.202,50.629,160.010
C06018=1018.005,351.156,-148.547,171.210,50.627,160.011
C06019=1018.013,351.404,-148.583,171.218,50.624,160.011
C06020=1018.020,351.651,-148.621,171.225,50.622,160.012
C06021=1018.028,351.898,-148.658,171.233,50.620,160.013
C06022=1018.036,352.158,-148.697,171.241,50.617,160.013
C06023=1018.044,352.417,-148.736,171.249,50.615,160.014
C06024=1018.052,352.677,-148.775,171.257,50.612,160.015
C06025=1018.060,352.937,-148.815,171.266,50.610,160.016
C06026=1018.068,353.184,-148.852,171.274,50.607,160.017
C06027=1018.075,353.431,-148.889,171.281,50.605,160.017
C06028=1018.082,353.678,-148.927,171.290,50.603,160.018
C06029=1018.090,353.925,-148.964,171.297,50.600,160.019
C06030=1018.097,354.172,-149.001,171.305,50.598,160.020
C06031=1018.105,354.420,-149.039,171.313,50.595,160.021
C06032=1018.113,354.666,-149.077,171.321,50.593,160.021
C06033=1018.121,354.913,-149.114,171.329,50.591,160.022
C06034=1018.128,355.160,-149.152,171.337,50.589,160.023
C06035=1018.135,355.407,-149.189,171.344,50.586,160.024
C06036=1018.143,355.655,-149.228,171.353,50.584,160.025
C06037=1018.151,355.902,-149.265,171.361,50.582,160.026
C06038=1018.159,356.149,-149.302,171.369,50.580,160.026
C06039=1018.166,356.395,-149.341,171.377,50.578,160.027
C06040=1018.174,356.643,-149.379,171.385,50.575,160.028
C06041=1018.181,356.890,-149.416,171.392,50.573,160.029
C06042=1018.190,357.136,-149.454,171.401,50.571,160.030
C06043=1018.197,357.384,-149.492,171.409,50.569,160.031
C06044=1018.205,357.631,-149.530,171.417,50.567,160.031
C06045=1018.212,357.878,-149.567,171.425,50.565,160.032
C06046=1018.220,358.125,-149.606,171.433,50.563,160.033
C06047=1018.228,358.371,-149.644,171.441,50.561,160.034
C06048=1018.236,358.618,-149.681,171.449,50.558,160.035
C06049=1018.244,358.865,-149.720,171.457,50.556,160.036
C06050=1018.252,359.112,-149.758,171.466,50.554,160.037
C06051=1018.260,359.360,-149.796,171.473,50.552,160.038
C06052=1018.267,359.606,-149.834,171.482,50.550,160.039
C06053=1018.275,359.854,-149.873,171.490,50.548,160.040
C06054=1018.283,360.100,-149.911,171.498,50.547,160.040
C06055=1018.290,360.347,-149.949,171.506,50.544,160.041
C06056=1018.298,360.594,-149.988,171.515,50.542,160.042
C06057=1018.305,360.841,-150.027,171.523,50.541,160.043
C06058=1018.313,361.088,-150.065,171.531,50.539,160.044
C06059=1018.321,361.334,-150.104,171.539,50.537,160.045
C06060=1018.329,361.582,-150.142,171.548,50.535,160.046
C06061=1018.337,361.829,-150.181,171.556,50.533,160.047
C06062=1018.345,362.075,-150.219,171.564,50.532,160.048
C06063=1018.353,362.323,-150.258,171.573,50.529,160.049
C06064=1018.361,362.569,-150.296,171.581,50.527,160.050
C06065=1018.369,362.816,-150.334,171.590,50.526,160.051
C06066=1018.376,363.063,-150.373,171.598,50.523,160.052
C06067=1018.384,363.310,-150.413,171.606,50.522,160.053
C06068=1018.392,363.557,-150.451,171.614,50.520,160.054
C06069=1018.400,363.803,-150.489,171.623,50.518,160.055
C06070=1018.408,364.051,-150.528,171.632,50.517,160.056
C06071=1018.416,364.297,-150.567,171.640,50.514,160.057
C06072=1018.424,364.544,-150.606,171.649,50.513,160.058
C06073=1018.432,364.791,-150.644,171.656,50.511,160.059
C06074=1018.440,365.038,-150.684,171.665,50.509,160.060
C06075=1018.449,365.285,-150.722,171.674,50.508,160.061
C06076=1018.457,365.531,-150.762,171.682,50.506,160.062
C06077=1018.464,365.778,-150.800,171.691,50.504,160.063
C06078=1018.472,366.025,-150.840,171.700,50.502,160.064
C06079=1018.480,366.272,-150.878,171.709,50.501,160.065
C06080=1018.489,366.519,-150.918,171.718,50.499,160.066
C06081=1018.497,366.766,-150.956,171.726,50.497,160.067
C06082=1018.506,367.033,-150.999,171.735,50.495,160.068
C06083=1018.515,367.300,-151.041,171.745,50.494,160.070
C06084=1018.524,367.567,-151.083,171.753,50.492,160.071
C06085=1018.533,367.834,-151.126,171.764,50.491,160.072
C06086=1018.540,368.081,-151.166,171.772,50.489,160.073
C06087=1018.549,368.328,-151.205,171.781,50.487,160.074
C06088=1018.556,368.575,-151.244,171.790,50.486,160.076
C06089=1018.565,368.822,-151.284,171.799,50.484,160.077
C06090=1018.573,369.068,-151.323,171.807,50.483,160.078
C06091=1018.581,369.315,-151.363,171.816,50.481,160.079
C06092=1018.589,369.562,-151.402,171.825,50.479,160.080
C06093=1018.597,369.809,-151.442,171.834,50.478,160.081
C06094=1018.606,370.055,-151.482,171.843,50.477,160.082
C06095=1018.614,370.302,-151.522,171.852,50.475,160.083
C06096=1018.622,370.548,-151.562,171.861,50.474,160.085
C06097=1018.630,370.795,-151.601,171.870,50.473,160.086
C06098=1018.638,371.042,-151.641,171.878,50.471,160.087
C06099=1018.647,371.288,-151.680,171.887,50.470,160.088
C06100=1018.655,371.535,-151.721,171.896,50.469,160.089
C06101=1018.663,371.781,-151.760,171.905,50.467,160.091
C06102=1018.671,372.029,-151.800,171.914,50.465,160.092
C06103=1018.680,372.275,-151.840,171.923,50.464,160.093
C06104=1018.688,372.522,-151.880,171.932,50.463,160.094
C06105=1018.696,372.768,-151.920,171.941,50.462,160.095
C06106=1018.705,373.014,-151.960,171.950,50.460,160.097
C06107=1018.713,373.262,-152.000,171.959,50.459,160.098
C06108=1018.722,373.508,-152.040,171.968,50.458,160.099
C06109=1018.730,373.755,-152.080,171.977,50.457,160.100
C06110=1018.739,374.001,-152.120,171.987,50.455,160.102
C06111=1018.747,374.248,-152.160,171.996,50.454,160.103
C06112=1018.756,374.494,-152.200,172.005,50.453,160.104
C06113=1018.764,374.741,-152.240,172.014,50.452,160.105
C06114=1018.773,374.988,-152.281,172.023,50.450,160.106
C06115=1018.782,375.234,-152.321,172.032,50.449,160.108
C06116=1018.790,375.482,-152.361,172.042,50.448,160.109
C06117=1018.799,375.727,-152.401,172.052,50.447,160.111
C06118=1018.807,375.974,-152.442,172.060,50.445,160.112
C06119=1018.815,376.221,-152.483,172.070,50.444,160.113
C06120=1018.824,376.467,-152.523,172.079,50.443,160.114
C06121=1018.833,376.714,-152.564,172.088,50.442,160.116
C06122=1018.841,376.960,-152.604,172.098,50.441,160.117
C06123=1018.849,377.207,-152.645,172.107,50.440,160.118
C06124=1018.857,377.453,-152.686,172.116,50.439,160.120
C06125=1018.867,377.700,-152.726,172.126,50.438,160.121
C06126=1018.875,377.946,-152.767,172.136,50.436,160.122
C06127=1018.883,378.193,-152.808,172.145,50.436,160.124
C06128=1018.892,378.439,-152.849,172.154,50.435,160.125
C06129=1018.901,378.686,-152.890,172.164,50.434,160.127
C06130=1018.909,378.932,-152.930,172.174,50.433,160.128
C06131=1018.918,379.179,-152.971,172.183,50.432,160.129
C06132=1018.926,379.424,-153.013,172.192,50.431,160.131
C06133=1018.935,379.671,-153.054,172.202,50.430,160.132
C06134=1018.944,379.918,-153.094,172.212,50.429,160.133
C06135=1018.952,380.164,-153.135,172.221,50.428,160.135
C06136=1018.961,380.411,-153.176,172.231,50.428,160.136
C06137=1018.970,380.657,-153.218,172.241,50.426,160.138
C06138=1018.979,380.904,-153.259,172.250,50.426,160.139
C06139=1018.988,381.149,-153.300,172.260,50.424,160.141
C06140=1018.996,381.396,-153.341,172.270,50.424,160.142
C06141=1019.005,381.643,-153.383,172.279,50.423,160.143
C06142=1019.016,381.932,-153.431,172.291,50.422,160.145
C06143=1019.026,382.222,-153.479,172.302,50.421,160.147
C06144=1019.036,382.511,-153.528,172.314,50.420,160.149
C06145=1019.047,382.801,-153.576,172.326,50.419,160.150
C06146=1019.056,383.047,-153.618,172.335,50.418,160.152
C06147=1019.065,383.293,-153.660,172.345,50.417,160.153
C06148=1019.074,383.540,-153.700,172.355,50.417,160.155
C06149=1019.083,383.786,-153.742,172.365,50.416,160.156
C06150=1019.092,384.033,-153.784,172.375,50.415,160.158
C06151=1019.101,384.279,-153.825,172.385,50.414,160.159
C06152=1019.110,384.525,-153.867,172.395,50.414,160.161
C06153=1019.120,384.771,-153.908,172.405,50.413,160.163
C06154=1019.129,385.018,-153.950,172.416,50.412,160.164
C06155=1019.137,385.264,-153.992,172.425,50.411,160.166
C06156=1019.146,385.511,-154.033,172.436,50.411,160.167
C06157=1019.155,385.757,-154.075,172.445,50.410,160.169
C06158=1019.165,386.003,-154.118,172.456,50.410,160.170
C06159=1019.174,386.249,-154.159,172.465,50.409,160.172
C06160=1019.182,386.495,-154.201,172.476,50.409,160.174
C06161=1019.192,386.742,-154.244,172.486,50.409,160.175
C06162=1019.201,386.988,-154.285,172.496,50.408,160.177
C06163=1019.210,387.235,-154.327,172.507,50.407,160.178
C06164=1019.219,387.480,-154.370,172.516,50.407,160.180
C06165=1019.228,387.727,-154.411,172.527,50.406,160.181
C06166=1019.238,387.972,-154.454,172.538,50.406,160.183
C06167=1019.247,388.219,-154.496,172.547,50.405,160.185
C06168=1019.256,388.466,-154.539,172.558,50.404,160.186
C06169=1019.265,388.711,-154.581,172.569,50.404,160.188
C06170=1019.274,388.958,-154.623,172.579,50.404,160.190
C06171=1019.284,389.204,-154.666,172.589,50.404,160.192
C06172=1019.293,389.450,-154.708,172.600,50.403,160.193
C06173=1019.301,389.696,-154.751,172.610,50.403,160.195
C06174=1019.311,389.942,-154.794,172.620,50.402,160.197
C06175=1019.320,390.188,-154.837,172.631,50.402,160.198
C06176=1019.329,390.434,-154.878,172.642,50.401,160.200
C06177=1019.339,390.681,-154.921,172.653,50.401,160.202
C06178=1019.348,390.927,-154.964,172.663,50.401,160.204
C06179=1019.358,391.173,-155.007,172.673,50.400,160.205
C06180=1019.367,391.419,-155.049,172.684,50.400,160.207
C06181=1019.377,391.666,-155.092,172.695,50.400,160.209
C06182=1019.386,391.911,-155.135,172.706,50.400,160.211
C06183=1019.395,392.157,-155.179,172.716,50.399,160.212
C06184=1019.405,392.403,-155.221,172.727,50.399,160.214
C06185=1019.414,392.650,-155.264,172.738,50.399,160.216
C06186=1019.423,392.895,-155.308,172.749,50.399,160.218
C06187=1019.433,393.142,-155.350,172.760,50.399,160.219
C06188=1019.443,393.388,-155.393,172.770,50.398,160.221
C06189=1019.452,393.633,-155.437,172.781,50.398,160.223
C06190=1019.461,393.880,-155.480,172.792,50.398,160.225
C06191=1019.471,394.125,-155.523,172.803,50.398,160.227
C06192=1019.480,394.372,-155.566,172.814,50.398,160.229
C06193=1019.490,394.618,-155.610,172.825,50.397,160.230
C06194=1019.499,394.864,-155.653,172.835,50.398,160.232
C06195=1019.509,395.109,-155.696,172.846,50.398,160.234
C06196=1019.519,395.355,-155.740,172.858,50.397,160.236
C06197=1019.528,395.602,-155.783,172.869,50.397,160.238
C06198=1019.538,395.848,-155.827,172.881,50.397,160.240
C06199=1019.548,396.093,-155.870,172.892,50.397,160.242
C06200=1019.557,396.339,-155.914,172.902,50.397,160.244
C06201=1019.567,396.585,-155.958,172.914,50.397,160.246
C06202=1019.581,396.912,-156.015,172.929,50.397,160.248
C06203=1019.593,397.240,-156.074,172.943,50.397,160.251
C06204=1019.606,397.566,-156.132,172.958,50.398,160.253
C06205=1019.620,397.894,-156.190,172.973,50.398,160.256
C06206=1019.629,398.140,-156.234,172.984,50.398,160.258
C06207=1019.639,398.386,-156.278,172.997,50.398,160.260
C06208=1019.649,398.631,-156.322,173.008,50.398,160.262
C06209=1019.659,398.877,-156.366,173.019,50.398,160.264
C06210=1019.668,399.123,-156.410,173.030,50.398,160.266
C06211=1019.678,399.369,-156.455,173.042,50.399,160.268
C06212=1019.688,399.615,-156.498,173.054,50.399,160.270
C06213=1019.698,399.861,-156.542,173.065,50.399,160.272
C06214=1019.708,400.106,-156.587,173.076,50.399,160.274
C06215=1019.718,400.352,-156.631,173.088,50.399,160.276
C06216=1019.727,400.597,-156.676,173.100,50.399,160.278
C06217=1019.738,400.843,-156.720,173.111,50.400,160.280
C06218=1019.748,401.090,-156.764,173.123,50.401,160.282
C06219=1019.757,401.335,-156.809,173.135,50.401,160.285
C06220=1019.767,401.581,-156.854,173.147,50.401,160.287
C06221=1019.777,401.826,-156.899,173.158,50.401,160.289
C06222=1019.788,402.073,-156.943,173.170,50.401,160.291
C06223=1019.797,402.318,-156.987,173.182,50.402,160.293
C06224=1019.807,402.564,-157.032,173.193,50.402,160.295
C06225=1019.817,402.810,-157.078,173.206,50.402,160.297
C06226=1019.828,403.055,-157.122,173.217,50.403,160.299
C06227=1019.837,403.301,-157.167,173.230,50.403,160.302
C06228=1019.848,403.547,-157.212,173.241,50.404,160.304
C06229=1019.858,403.792,-157.257,173.254,50.404,160.306
C06230=1019.868,404.039,-157.302,173.265,50.405,160.308
C06231=1019.879,404.283,-157.347,173.278,50.405,160.310
C06232=1019.889,404.529,-157.392,173.289,50.406,160.313
C06233=1019.899,404.775,-157.437,173.302,50.406,160.315
C06234=1019.909,405.021,-157.482,173.313,50.407,160.317
C06235=1019.920,405.266,-157.527,173.326,50.407,160.319
C06236=1019.930,405.512,-157.572,173.338,50.407,160.321
C06237=1019.940,405.757,-157.618,173.350,50.408,160.324
C06238=1019.950,406.003,-157.663,173.363,50.409,160.326
C06239=1019.961,406.249,-157.707,173.376,50.409,160.328
C06240=1019.971,406.494,-157.753,173.387,50.410,160.330
C06241=1019.982,406.739,-157.799,173.400,50.410,160.333
C06242=1019.992,406.986,-157.844,173.412,50.411,160.335
C06243=1020.003,407.231,-157.890,173.424,50.412,160.337
C06244=1020.013,407.476,-157.934,173.437,50.412,160.340
C06245=1020.024,407.722,-157.980,173.449,50.413,160.342
C06246=1020.035,407.968,-158.026,173.462,50.413,160.344
C06247=1020.045,408.213,-158.072,173.475,50.414,160.347
C06248=1020.056,408.459,-158.116,173.487,50.415,160.349
C06249=1020.067,408.705,-158.162,173.500,50.416,160.351
C06250=1020.078,408.950,-158.208,173.512,50.416,160.354
C06251=1020.088,409.196,-158.254,173.525,50.417,160.356
C06252=1020.099,409.441,-158.300,173.538,50.418,160.359
C06253=1020.110,409.686,-158.347,173.551,50.418,160.361
C06254=1020.120,409.932,-158.393,173.564,50.419,160.364
C06255=1020.130,410.178,-158.439,173.576,50.420,160.366
C06256=1020.141,410.423,-158.485,173.589,50.421,160.368
C06257=1020.152,410.668,-158.532,173.602,50.422,160.371
C06258=1020.162,410.914,-158.578,173.615,50.423,160.373
C06259=1020.173,411.160,-158.623,173.628,50.424,160.376
C06260=1020.184,411.405,-158.670,173.641,50.425,160.378
C06261=1020.195,411.650,-158.716,173.654,50.426,160.381
C06262=1020.208,411.941,-158.771,173.669,50.427,160.384
C06263=1020.220,412.231,-158.826,173.685,50.427,160.387
C06264=1020.233,412.522,-158.881,173.701,50.429,160.390
C06265=1020.246,412.813,-158.936,173.716,50.430,160.393
C06266=1020.257,413.058,-158.983,173.729,50.431,160.395
C06267=1020.269,413.303,-159.030,173.743,50.432,160.398
C06268=1020.280,413.548,-159.076,173.756,50.433,160.400
C06269=1020.290,413.793,-159.123,173.769,50.434,160.403
C06270=1020.302,414.039,-159.170,173.783,50.435,160.405
C06271=1020.312,414.285,-159.217,173.797,50.435,160.408
C06272=1020.323,414.530,-159.264,173.810,50.437,160.411
C06273=1020.334,414.775,-159.310,173.823,50.438,160.413
C06274=1020.346,415.021,-159.357,173.836,50.439,160.416
C06275=1020.357,415.265,-159.405,173.850,50.440,160.419
C06276=1020.368,415.511,-159.452,173.864,50.441,160.421
C06277=1020.379,415.756,-159.499,173.877,50.443,160.424
C06278=1020.391,416.001,-159.546,173.892,50.444,160.427
C06279=1020.401,416.247,-159.594,173.905,50.445,160.429
C06280=1020.412,416.492,-159.641,173.919,50.446,160.432
C06281=1020.424,416.737,-159.688,173.932,50.447,160.435
C06282=1020.434,416.983,-159.736,173.947,50.448,160.438
C06283=1020.446,417.228,-159.783,173.960,50.450,160.440
C06284=1020.458,417.473,-159.831,173.975,50.451,160.443
C06285=1020.469,417.719,-159.879,173.988,50.452,160.446
C06286=1020.480,417.963,-159.926,174.002,50.453,160.449
C06287=1020.491,418.209,-159.974,174.016,50.455,160.451
C06288=1020.503,418.454,-160.021,174.030,50.456,160.454
C06289=1020.515,418.699,-160.069,174.045,50.457,160.457
C06290=1020.526,418.945,-160.117,174.058,50.459,160.460
C06291=1020.538,419.190,-160.165,174.073,50.460,160.463
C06292=1020.549,419.435,-160.213,174.087,50.461,160.466
C06293=1020.560,419.680,-160.261,174.101,50.463,160.468
C06294=1020.572,419.925,-160.309,174.115,50.464,160.471
C06295=1020.584,420.170,-160.356,174.130,50.466,160.474
C06296=1020.595,420.416,-160.405,174.145,50.467,160.477
C06297=1020.607,420.660,-160.453,174.158,50.469,160.480
C06298=1020.619,420.905,-160.501,174.173,50.470,160.483
C06299=1020.630,421.150,-160.549,174.188,50.471,160.486
C06300=1020.643,421.396,-160.597,174.202,50.473,160.489
C06301=1020.654,421.641,-160.646,174.217,50.474,160.492
C06302=1020.666,421.886,-160.694,174.231,50.476,160.495
C06303=1020.677,422.131,-160.743,174.246,50.477,160.498
C06304=1020.689,422.375,-160.792,174.261,50.479,160.501
C06305=1020.701,422.621,-160.840,174.276,50.480,160.504
C06306=1020.713,422.866,-160.889,174.291,50.482,160.507
C06307=1020.725,423.110,-160.937,174.305,50.484,160.510
C06308=1020.737,423.356,-160.987,174.320,50.485,160.513
C06309=1020.749,423.601,-161.034,174.335,50.487,160.516
C06310=1020.760,423.846,-161.083,174.350,50.489,160.519
C06311=1020.772,424.091,-161.133,174.365,50.490,160.522
C06312=1020.784,424.336,-161.181,174.381,50.492,160.525
C06313=1020.796,424.581,-161.231,174.396,50.493,160.528
C06314=1020.808,424.825,-161.279,174.411,50.495,160.532
C06315=1020.820,425.071,-161.328,174.426,50.497,160.535
C06316=1020.833,425.316,-161.378,174.442,50.499,160.538
C06317=1020.845,425.560,-161.427,174.457,50.500,160.541
C06318=1020.857,425.806,-161.476,174.472,50.502,160.544
C06319=1020.869,426.050,-161.526,174.488,50.504,160.548
C06320=1020.881,426.295,-161.575,174.503,50.506,160.551
C06321=1020.893,426.540,-161.625,174.518,50.508,160.554
C06322=1020.515,424.580,-161.567,174.384,50.563,160.547
C06323=1020.503,424.334,-161.518,174.368,50.562,160.543
C06324=1020.491,424.090,-161.470,174.353,50.560,160.540
C06325=1020.479,423.844,-161.420,174.338,50.558,160.537
C06326=1020.466,423.600,-161.372,174.323,50.557,160.534
C06327=1020.455,423.354,-161.323,174.307,50.555,160.531
C06328=1020.443,423.109,-161.274,174.293,50.554,160.528
C06329=1020.431,422.865,-161.226,174.278,50.552,160.525
C06330=1020.419,422.619,-161.176,174.263,50.551,160.522
C06331=1020.407,422.374,-161.129,174.248,50.550,160.519
C06332=1020.396,422.130,-161.080,174.233,50.548,160.516
C06333=1020.384,421.885,-161.031,174.219,50.547,160.513
C06334=1020.373,421.640,-160.983,174.204,50.545,160.510
C06335=1020.360,421.395,-160.934,174.190,50.544,160.507
C06336=1020.349,421.149,-160.886,174.175,50.542,160.504
C06337=1020.337,420.904,-160.838,174.160,50.541,160.501
C06338=1020.326,420.659,-160.790,174.146,50.540,160.498
C06339=1020.314,420.414,-160.741,174.131,50.539,160.495
C06340=1020.302,420.169,-160.694,174.117,50.537,160.493
C06341=1020.291,419.924,-160.645,174.102,50.536,160.489
C06342=1020.279,419.679,-160.598,174.088,50.534,160.487
C06343=1020.268,419.434,-160.549,174.074,50.533,160.484
C06344=1020.256,419.189,-160.502,174.059,50.532,160.481
C06345=1020.244,418.943,-160.454,174.045,50.531,160.478
C06346=1020.233,418.698,-160.406,174.031,50.530,160.475
C06347=1020.222,418.452,-160.359,174.017,50.528,160.473
C06348=1020.210,418.207,-160.311,174.003,50.527,160.470
C06349=1020.199,417.962,-160.263,173.988,50.526,160.467
C06350=1020.188,417.717,-160.216,173.975,50.525,160.464
C06351=1020.176,417.472,-160.168,173.960,50.524,160.461
C06352=1020.165,417.227,-160.120,173.946,50.523,160.459
C06353=1020.153,416.981,-160.073,173.933,50.522,160.456
C06354=1020.142,416.737,-160.026,173.918,50.520,160.453
C06355=1020.131,416.491,-159.978,173.905,50.519,160.451
C06356=1020.119,416.246,-159.930,173.891,50.518,160.448
C06357=1020.108,416.001,-159.884,173.878,50.517,160.445
C06358=1020.098,415.755,-159.836,173.864,50.516,160.443
C06359=1020.086,415.510,-159.789,173.850,50.515,160.440
C06360=1020.075,415.265,-159.742,173.837,50.514,160.437
C06361=1020.065,415.019,-159.695,173.823,50.513,160.435
C06362=1020.053,414.774,-159.648,173.810,50.512,160.432
C06363=1020.042,414.529,-159.601,173.795,50.511,160.429
C06364=1020.031,414.283,-159.554,173.782,50.510,160.427
C06365=1020.020,414.038,-159.507,173.769,50.509,160.424
C06366=1020.008,413.792,-159.460,173.755,50.508,160.421
C06367=1019.997,413.547,-159.414,173.742,50.507,160.419
C06368=1019.986,413.302,-159.367,173.729,50.507,160.416
C06369=1019.976,413.056,-159.320,173.715,50.506,160.414
C06370=1019.965,412.811,-159.274,173.702,50.505,160.411
C06371=1019.953,412.544,-159.224,173.687,50.504,160.408
C06372=1019.941,412.277,-159.173,173.673,50.503,160.406
C06373=1019.929,412.011,-159.123,173.659,50.502,160.403
C06374=1019.917,411.745,-159.072,173.644,50.501,160.400
C06375=1019.907,411.498,-159.025,173.632,50.501,160.398
C06376=1019.896,411.253,-158.979,173.619,50.500,160.395
C06377=1019.885,411.008,-158.933,173.606,50.499,160.393
C06378=1019.874,410.763,-158.886,173.593,50.498,160.390
C06379=1019.864,410.517,-158.840,173.580,50.498,160.388
C06380=1019.853,410.272,-158.794,173.567,50.496,160.385
C06381=1019.842,410.026,-158.749,173.554,50.496,160.383
C06382=1019.831,409.781,-158.702,173.542,50.495,160.381
C06383=1019.821,409.536,-158.656,173.528,50.494,160.378
C06384=1019.810,409.290,-158.610,173.516,50.494,160.376
C06385=1019.800,409.044,-158.564,173.503,50.493,160.374
C06386=1019.790,408.798,-158.518,173.490,50.493,160.371
C06387=1019.778,408.553,-158.472,173.478,50.492,160.369
C06388=1019.768,408.308,-158.427,173.464,50.491,160.366
C06389=1019.758,408.062,-158.382,173.452,50.491,160.364
C06390=1019.747,407.816,-158.336,173.439,50.491,160.362
C06391=1019.736,407.571,-158.290,173.427,50.490,160.359
C06392=1019.725,407.326,-158.245,173.414,50.490,160.357
C06393=1019.715,407.079,-158.199,173.402,50.489,160.355
C06394=1019.705,406.835,-158.154,173.389,50.488,160.353
C06395=1019.694,406.589,-158.109,173.377,50.488,160.350
C06396=1019.683,406.343,-158.063,173.364,50.487,160.348
C06397=1019.673,406.097,-158.018,173.353,50.487,160.346
C06398=1019.663,405.852,-157.973,173.340,50.487,160.343
C06399=1019.652,405.606,-157.928,173.327,50.486,160.341
C06400=1019.642,405.361,-157.882,173.315,50.486,160.339
C06401=1019.632,405.115,-157.837,173.303,50.485,160.337
C06402=1019.622,404.869,-157.792,173.291,50.485,160.335
C06403=1019.612,404.623,-157.747,173.278,50.485,160.332
C06404=1019.600,404.378,-157.702,173.267,50.484,160.330
C06405=1019.591,404.132,-157.657,173.254,50.484,160.328
C06406=1019.581,403.887,-157.612,173.243,50.484,160.326
C06407=1019.571,403.641,-157.567,173.230,50.484,160.324
C06408=1019.560,403.395,-157.523,173.218,50.483,160.321
C06409=1019.550,403.149,-157.478,173.206,50.483,160.319
C06410=1019.540,402.904,-157.433,173.194,50.483,160.317
C06411=1019.530,402.658,-157.388,173.182,50.482,160.315
C06412=1019.519,402.412,-157.343,173.170,50.482,160.313
C06413=1019.510,402.167,-157.299,173.159,50.482,160.311
C06414=1019.500,401.921,-157.254,173.147,50.481,160.309
C06415=1019.490,401.676,-157.209,173.135,50.481,160.307
C06416=1019.479,401.429,-157.165,173.124,50.481,160.304
C06417=1019.470,401.184,-157.120,173.111,50.481,160.302
C06418=1019.460,400.938,-157.075,173.100,50.481,160.300
C06419=1019.451,400.692,-157.031,173.088,50.481,160.298
C06420=1019.440,400.447,-156.987,173.076,50.480,160.296
C06421=1019.431,400.201,-156.943,173.065,50.480,160.294
C06422=1019.420,399.955,-156.898,173.053,50.480,160.292
C06423=1019.410,399.709,-156.854,173.041,50.480,160.290
C06424=1019.401,399.463,-156.809,173.030,50.480,160.288
C06425=1019.390,399.217,-156.766,173.018,50.480,160.286
C06426=1019.381,398.971,-156.722,173.007,50.480,160.284
C06427=1019.371,398.726,-156.677,172.996,50.480,160.282
C06428=1019.361,398.480,-156.634,172.984,50.480,160.280
C06429=1019.352,398.234,-156.589,172.972,50.480,160.278
C06430=1019.342,397.988,-156.546,172.961,50.480,160.276
C06431=1019.329,397.658,-156.487,172.946,50.479,160.273
C06432=1019.315,397.329,-156.428,172.930,50.480,160.271
C06433=1019.303,397.000,-156.370,172.916,50.480,160.268
C06434=1019.289,396.670,-156.311,172.901,50.480,160.266
C06435=1019.280,396.424,-156.267,172.890,50.480,160.264
C06436=1019.270,396.178,-156.224,172.879,50.480,160.262
C06437=1019.260,395.933,-156.180,172.867,50.481,160.260
C06438=1019.251,395.686,-156.137,172.856,50.481,160.258
C06439=1019.241,395.441,-156.094,172.845,50.481,160.256
C06440=1019.231,395.195,-156.050,172.833,50.481,160.254
C06441=1019.222,394.948,-156.007,172.822,50.481,160.252
C06442=1019.212,394.703,-155.964,172.812,50.481,160.251
C06443=1019.202,394.457,-155.921,172.801,50.481,160.249
C06444=1019.193,394.210,-155.877,172.790,50.482,160.247
C06445=1019.184,393.965,-155.834,172.779,50.482,160.245
C06446=1019.174,393.719,-155.790,172.768,50.482,160.243
C06447=1019.165,393.473,-155.748,172.757,50.482,160.241
C06448=1019.155,393.227,-155.704,172.746,50.482,160.240
C06449=1019.146,392.980,-155.661,172.735,50.483,160.238
C06450=1019.137,392.734,-155.618,172.724,50.483,160.236
C06451=1019.127,392.489,-155.575,172.713,50.484,160.234
C06452=1019.118,392.243,-155.532,172.702,50.484,160.232
C06453=1019.108,391.996,-155.489,172.692,50.484,160.231
C06454=1019.099,391.750,-155.447,172.681,50.485,160.229
C06455=1019.089,391.504,-155.404,172.670,50.485,160.227
C06456=1019.080,391.258,-155.361,172.659,50.485,160.225
C06457=1019.071,391.011,-155.318,172.650,50.486,160.224
C06458=1019.061,390.766,-155.276,172.639,50.486,160.222
C06459=1019.052,390.519,-155.233,172.628,50.487,160.220
C06460=1019.042,390.274,-155.190,172.617,50.487,160.219
C06461=1019.033,390.028,-155.148,172.607,50.488,160.217
C06462=1019.024,389.781,-155.105,172.596,50.488,160.215
C06463=1019.015,389.535,-155.062,172.586,50.488,160.214
C06464=1019.006,389.289,-155.020,172.575,50.489,160.212
C06465=1018.997,389.043,-154.978,172.564,50.489,160.210
C06466=1018.987,388.797,-154.935,172.554,50.490,160.208
C06467=1018.979,388.550,-154.893,172.544,50.490,160.207
C06468=1018.969,388.304,-154.850,172.533,50.491,160.205
C06469=1018.960,388.059,-154.808,172.523,50.492,160.203
C06470=1018.951,387.811,-154.766,172.512,50.492,160.202
C06471=1018.941,387.566,-154.724,172.503,50.493,160.200
C06472=1018.932,387.319,-154.682,172.492,50.494,160.199
C06473=1018.924,387.073,-154.640,172.481,50.494,160.197
C06474=1018.914,386.827,-154.598,172.472,50.494,160.195
C06475=1018.905,386.581,-154.556,172.461,50.495,160.194
C06476=1018.896,386.334,-154.514,172.451,50.496,160.192
C06477=1018.887,386.088,-154.471,172.441,50.496,160.191
C06478=1018.878,385.842,-154.430,172.430,50.497,160.189
C06479=1018.869,385.595,-154.388,172.420,50.498,160.187
C06480=1018.860,385.349,-154.346,172.411,50.499,160.186
C06481=1018.851,385.103,-154.304,172.400,50.500,160.184
C06482=1018.842,384.857,-154.262,172.390,50.500,160.183
C06483=1018.833,384.610,-154.221,172.380,50.501,160.181
C06484=1018.824,384.364,-154.179,172.370,50.502,160.180
C06485=1018.814,384.117,-154.138,172.360,50.503,160.178
C06486=1018.805,383.871,-154.097,172.350,50.503,160.177
C06487=1018.796,383.625,-154.055,172.341,50.504,160.175
C06488=1018.788,383.378,-154.013,172.330,50.505,160.174
C06489=1018.778,383.132,-153.972,172.319,50.506,160.172
C06490=1018.770,382.886,-153.931,172.310,50.507,160.171
C06491=1018.759,382.595,-153.881,172.299,50.508,160.169
C06492=1018.749,382.303,-153.833,172.287,50.509,160.167
C06493=1018.738,382.011,-153.784,172.275,50.510,160.165
C06494=1018.728,381.719,-153.735,172.264,50.511,160.164
C06495=1018.719,381.472,-153.694,172.254,50.512,160.162
C06496=1018.709,381.226,-153.653,172.244,50.513,160.161
C06497=1018.701,380.980,-153.612,172.234,50.514,160.159
C06498=1018.692,380.733,-153.571,172.225,50.515,160.158
C06499=1018.684,380.486,-153.530,172.214,50.517,160.157
C06500=1018.675,380.240,-153.488,172.205,50.517,160.155
C06501=1018.666,379.994,-153.448,172.196,50.518,160.154
C06502=1018.657,379.748,-153.406,172.186,50.519,160.152
C06503=1018.648,379.501,-153.365,172.176,50.520,160.151
C06504=1018.640,379.254,-153.325,172.166,50.522,160.150
C06505=1018.631,379.008,-153.283,172.157,50.522,160.148
C06506=1018.623,378.762,-153.243,172.147,50.523,160.147
C06507=1018.614,378.515,-153.202,172.137,50.525,160.145
C06508=1018.606,378.269,-153.161,172.128,50.526,160.144
C06509=1018.597,378.022,-153.120,172.119,50.527,160.143
C06510=1018.589,377.776,-153.080,172.109,50.528,160.141
C06511=1018.580,377.529,-153.038,172.100,50.529,160.140
C06512=1018.572,377.283,-152.998,172.090,50.530,160.139
C06513=1018.563,377.036,-152.957,172.080,50.531,160.137
C06514=1018.554,376.790,-152.917,172.071,50.532,160.136
C06515=1018.546,376.543,-152.876,172.062,50.533,160.135
C06516=1018.538,376.297,-152.835,172.053,50.535,160.134
C06517=1018.530,376.051,-152.794,172.043,50.536,160.132
C06518=1018.521,375.803,-152.755,172.034,50.537,160.131
C06519=1018.513,375.557,-152.714,172.025,50.538,160.130
C06520=1018.503,375.310,-152.674,172.016,50.540,160.128
C06521=1018.495,375.064,-152.633,172.006,50.541,160.127
C06522=1018.487,374.817,-152.594,171.997,50.542,160.126
C06523=1018.478,374.570,-152.553,171.988,50.544,160.125
C06524=1018.470,374.324,-152.513,171.979,50.545,160.123
C06525=1018.462,374.078,-152.473,171.970,50.547,160.122
C06526=1018.453,373.830,-152.433,171.960,50.548,160.121
C06527=1018.444,373.584,-152.393,171.951,50.550,160.120
C06528=1018.436,373.337,-152.353,171.942,50.551,160.118
C06529=1018.427,373.091,-152.313,171.933,50.552,160.117
C06530=1018.419,372.844,-152.273,171.924,50.553,160.116
C06531=1018.410,372.598,-152.233,171.914,50.555,160.115
C06532=1018.402,372.351,-152.193,171.905,50.557,160.114
C06533=1018.394,372.104,-152.154,171.896,50.558,160.112
C06534=1018.386,371.858,-152.114,171.887,50.559,160.111
C06535=1018.378,371.611,-152.074,171.878,50.561,160.110
C06536=1018.368,371.364,-152.034,171.869,50.562,160.109
C06537=1018.361,371.117,-151.994,171.860,50.564,160.108
C06538=1018.352,370.871,-151.955,171.852,50.565,160.106
C06539=1018.345,370.624,-151.915,171.842,50.567,160.105
C06540=1018.336,370.378,-151.875,171.833,50.569,160.104
C06541=1018.327,370.131,-151.835,171.824,50.570,160.103
C06542=1018.320,369.884,-151.795,171.815,50.571,160.102
C06543=1018.311,369.638,-151.756,171.806,50.573,160.101
C06544=1018.303,369.391,-151.716,171.798,50.575,160.099
C06545=1018.295,369.144,-151.677,171.789,50.576,160.098
C06546=1018.287,368.897,-151.637,171.780,50.578,160.097
C06547=1018.279,368.651,-151.598,171.771,50.579,160.096
C06548=1018.270,368.404,-151.558,171.762,50.581,160.095
C06549=1018.263,368.157,-151.518,171.754,50.583,160.094
C06550=1018.255,367.911,-151.480,171.745,50.584,160.093
C06551=1018.247,367.641,-151.436,171.735,50.586,160.092
C06552=1018.238,367.371,-151.393,171.726,50.588,160.090
C06553=1018.228,367.102,-151.351,171.716,50.590,160.089
C06554=1018.219,366.832,-151.309,171.707,50.592,160.088
C06555=1018.211,366.586,-151.269,171.698,50.593,160.087
C06556=1018.203,366.339,-151.231,171.690,50.596,160.086
C06557=1018.195,366.092,-151.191,171.681,50.597,160.085
C06558=1018.187,365.845,-151.153,171.672,50.599,160.084
C06559=1018.179,365.598,-151.113,171.664,50.601,160.083
C06560=1018.171,365.351,-151.075,171.655,50.603,160.082
C06561=1018.163,365.105,-151.036,171.646,50.604,160.081
C06562=1018.155,364.858,-150.997,171.638,50.606,160.080
C06563=1018.147,364.611,-150.958,171.629,50.608,160.079
C06564=1018.138,364.364,-150.919,171.621,50.610,160.078
C06565=1018.131,364.118,-150.881,171.613,50.611,160.077
C06566=1018.122,363.870,-150.842,171.604,50.614,160.076
C06567=1018.115,363.623,-150.803,171.595,50.615,160.075
C06568=1018.107,363.377,-150.764,171.587,50.618,160.074
C06569=1018.099,363.130,-150.726,171.579,50.620,160.073
C06570=1018.091,362.883,-150.687,171.570,50.621,160.072
C06571=1018.083,362.636,-150.649,171.561,50.624,160.071
C06572=1018.075,362.389,-150.610,171.553,50.625,160.070
C06573=1018.068,362.142,-150.572,171.545,50.627,160.069
C06574=1018.059,361.895,-150.533,171.537,50.629,160.068
C06575=1018.052,361.649,-150.495,171.528,50.631,160.067
C06576=1018.044,361.401,-150.456,171.520,50.633,160.066
C06577=1018.036,361.155,-150.418,171.511,50.635,160.065
C06578=1018.029,360.907,-150.379,171.503,50.638,160.064
C06579=1018.021,360.661,-150.341,171.495,50.639,160.063
C06580=1018.013,360.414,-150.302,171.487,50.641,160.062
C06581=1018.006,360.167,-150.264,171.478,50.643,160.061
C06582=1017.997,359.920,-150.225,171.470,50.645,160.060
C06583=1017.990,359.673,-150.187,171.461,50.648,160.059
C06584=1017.982,359.426,-150.148,171.454,50.650,160.059
C06585=1017.974,359.179,-150.111,171.446,50.652,160.058
C06586=1017.967,358.933,-150.073,171.437,50.654,160.057
C06587=1017.959,358.685,-150.034,171.429,50.656,160.056
C06588=1017.951,358.438,-149.996,171.420,50.658,160.055
C06589=1017.943,358.191,-149.958,171.413,50.660,160.054
C06590=1017.935,357.944,-149.921,171.405,50.663,160.053
C06591=1017.928,357.698,-149.883,171.396,50.665,160.052
C06592=1017.920,357.450,-149.845,171.388,50.667,160.051
C06593=1017.912,357.203,-149.807,171.381,50.669,160.051
C06594=1017.905,356.956,-149.769,171.373,50.672,160.050
C06595=1017.896,356.709,-149.731,171.364,50.674,160.049
C06596=1017.889,356.462,-149.693,171.356,50.676,160.048
C06597=1017.882,356.215,-149.656,171.348,50.678,160.047
C06598=1017.874,355.968,-149.618,171.340,50.681,160.047
C06599=1017.866,355.721,-149.580,171.332,50.683,160.046
C06600=1017.858,355.474,-149.543,171.323,50.685,160.045
C06601=1017.851,355.227,-149.505,171.316,50.688,160.044
C06602=1017.844,354.980,-149.467,171.308,50.690,160.043
C06603=1017.836,354.733,-149.430,171.300,50.693,160.043
C06604=1017.828,354.486,-149.393,171.292,50.695,160.042
C06605=1017.821,354.238,-149.355,171.284,50.697,160.041
C06606=1017.813,353.992,-149.317,171.276,50.700,160.040
C06607=1017.806,353.745,-149.279,171.268,50.702,160.039
C06608=1017.798,353.498,-149.242,171.261,50.704,160.039
C06609=1017.791,353.251,-149.205,171.252,50.707,160.038
C06610=1017.783,353.004,-149.168,171.244,50.710,160.037
C06611=1017.775,352.741,-149.128,171.236,50.712,160.036
C06612=1017.767,352.479,-149.089,171.228,50.715,160.035
C06613=1017.759,352.218,-149.049,171.220,50.717,160.035
C06614=1017.750,351.956,-149.010,171.212,50.720,160.034
C06615=1017.743,351.709,-148.972,171.204,50.722,160.033
C06616=1017.736,351.461,-148.936,171.196,50.725,160.032
C06617=1017.728,351.214,-148.899,171.189,50.728,160.032
C06618=1017.721,350.967,-148.861,171.180,50.730,160.031
C06619=1017.713,350.720,-148.824,171.173,50.733,160.030
C06620=1017.706,350.472,-148.787,171.165,50.735,160.030
C06621=1017.698,350.226,-148.750,171.157,50.738,160.029
C06622=1017.691,349.978,-148.713,171.150,50.741,160.028
C06623=1017.683,349.731,-148.677,171.142,50.743,160.027
C06624=1017.676,349.484,-148.639,171.134,50.746,160.027
C06625=1017.669,349.237,-148.602,171.127,50.748,160.026
C06626=1017.661,348.989,-148.565,171.119,50.751,160.025
C06627=1017.654,348.743,-148.528,171.112,50.754,160.025
C06628=1017.647,348.495,-148.492,171.104,50.756,160.024
C06629=1017.640,348.248,-148.455,171.096,50.759,160.023
C06630=1017.632,348.001,-148.418,171.089,50.762,160.023
C06631=1017.625,347.754,-148.381,171.081,50.765,160.022
C06632=1017.618,347.507,-148.345,171.074,50.767,160.021
C06633=1017.610,347.260,-148.307,171.066,50.770,160.021
C06634=1017.603,347.012,-148.271,171.059,50.773,160.020
C06635=1017.596,346.765,-148.234,171.051,50.775,160.019
C06636=1017.589,346.518,-148.199,171.043,50.778,160.019
C06637=1017.581,346.271,-148.162,171.036,50.781,160.018
C06638=1017.574,346.023,-148.125,171.028,50.784,160.017
C06639=1017.566,345.776,-148.089,171.021,50.787,160.017
C06640=1017.559,345.529,-148.053,171.013,50.790,160.016
C06641=1017.552,345.281,-148.016,171.006,50.792,160.015
C06642=1017.544,345.034,-147.980,170.998,50.796,160.015
C06643=1017.537,344.787,-147.944,170.990,50.798,160.014
C06644=1017.530,344.540,-147.906,170.983,50.801,160.014
C06645=1017.522,344.293,-147.870,170.976,50.804,160.013
C06646=1017.515,344.046,-147.834,170.969,50.807,160.013
C06647=1017.508,343.798,-147.798,170.961,50.810,160.012
C06648=1017.501,343.551,-147.761,170.954,50.813,160.011
C06649=1017.494,343.304,-147.725,170.946,50.816,160.011
C06650=1017.486,343.056,-147.690,170.940,50.819,160.010
C06651=1017.480,342.809,-147.653,170.932,50.822,160.010
C06652=1017.472,342.561,-147.617,170.925,50.825,160.009
C06653=1017.465,342.315,-147.581,170.917,50.828,160.008
C06654=1017.457,342.067,-147.545,170.910,50.831,160.008
C06655=1017.451,341.820,-147.509,170.902,50.834,160.007
C06656=1017.444,341.572,-147.473,170.896,50.837,160.007
C06657=1017.437,341.325,-147.437,170.888,50.840,160.006
C06658=1017.429,341.078,-147.401,170.881,50.843,160.006
C06659=1017.423,340.831,-147.365,170.873,50.846,160.005
C06660=1017.415,340.583,-147.329,170.866,50.849,160.005
C06661=1017.408,340.336,-147.293,170.859,50.852,160.004
C06662=1017.400,340.088,-147.257,170.852,50.855,160.004
C06663=1017.394,339.841,-147.222,170.844,50.858,160.003
C06664=1017.387,339.594,-147.186,170.838,50.861,160.003
C06665=1017.380,339.346,-147.150,170.830,50.865,160.002
C06666=1017.373,339.099,-147.114,170.823,50.867,160.001
C06667=1017.366,338.851,-147.079,170.815,50.871,160.001
C06668=1017.359,338.604,-147.043,170.809,50.874,160.001
C06669=1017.352,338.357,-147.008,170.801,50.877,160.000
C06670=1017.344,338.110,-146.971,170.794,50.881,160.000
C06671=1017.336,337.845,-146.934,170.787,50.884,159.999
C06672=1017.329,337.580,-146.896,170.779,50.888,159.999
C06673=1017.322,337.316,-146.858,170.772,50.891,159.998
C06674=1017.314,337.051,-146.820,170.764,50.895,159.998
C06675=1017.307,336.804,-146.785,170.756,50.898,159.997
C06676=1017.300,336.555,-146.750,170.750,50.901,159.997
C06677=1017.293,336.309,-146.714,170.743,50.904,159.996
C06678=1017.286,336.061,-146.679,170.736,50.908,159.996
C06679=1017.279,335.814,-146.644,170.729,50.911,159.995
C06680=1017.272,335.566,-146.608,170.721,50.914,159.995
C06681=1017.265,335.319,-146.573,170.715,50.918,159.994
C06682=1017.258,335.071,-146.538,170.707,50.921,159.994
C06683=1017.252,334.824,-146.503,170.701,50.924,159.994
C06684=1017.245,334.576,-146.468,170.693,50.928,159.993
C06685=1017.237,334.328,-146.432,170.687,50.932,159.993
C06686=1017.231,334.081,-146.397,170.680,50.935,159.992
C06687=1017.224,333.834,-146.361,170.672,50.938,159.992
C06688=1017.216,333.587,-146.327,170.666,50.941,159.991
C06689=1017.210,333.339,-146.292,170.659,50.945,159.991
C06690=1017.203,333.092,-146.257,170.652,50.949,159.991
C06691=1017.196,332.845,-146.222,170.645,50.952,159.990
C06692=1017.189,332.597,-146.187,170.638,50.955,159.990
C06693=1017.183,332.350,-146.152,170.632,50.959,159.990
C06694=1017.176,332.102,-146.116,170.624,50.963,159.989
C06695=1017.168,331.855,-146.082,170.618,50.966,159.989
C06696=1017.161,331.607,-146.047,170.610,50.970,159.988
C06697=1017.154,331.359,-146.012,170.604,50.973,159.988
C06698=1017.148,331.112,-145.977,170.597,50.977,159.988
C06699=1017.141,330.864,-145.943,170.590,50.980,159.987
C06700=1017.134,330.617,-145.908,170.583,50.984,159.987
C06701=1017.127,330.370,-145.873,170.576,50.988,159.987
C06702=1017.120,330.122,-145.839,170.570,50.991,159.986
C06703=1017.113,329.874,-145.804,170.563,50.995,159.986
C06704=1017.107,329.627,-145.770,170.556,50.999,159.986
C06705=1017.100,329.380,-145.735,170.550,51.002,159.985
C06706=1017.093,329.132,-145.701,170.542,51.006,159.985
C06707=1017.086,328.885,-145.666,170.536,51.010,159.985
C06708=1017.079,328.637,-145.632,170.529,51.013,159.984
C06709=1017.072,328.390,-145.597,170.522,51.017,159.984
C06710=1017.066,328.142,-145.562,170.516,51.021,159.984
C06711=1017.059,327.894,-145.527,170.508,51.024,159.983
C06712=1017.052,327.647,-145.493,170.502,51.028,159.983
C06713=1017.046,327.399,-145.459,170.496,51.032,159.983
C06714=1017.039,327.152,-145.424,170.488,51.036,159.983
C06715=1017.032,326.904,-145.390,170.482,51.039,159.982
C06716=1017.026,326.656,-145.356,170.476,51.043,159.982
C06717=1017.019,326.409,-145.321,170.468,51.047,159.982
C06718=1017.012,326.162,-145.287,170.462,51.051,159.981
C06719=1017.006,325.914,-145.253,170.455,51.055,159.981
C06720=1016.999,325.666,-145.219,170.448,51.058,159.981
C06721=1016.991,325.419,-145.185,170.442,51.062,159.980
C06722=1016.985,325.172,-145.152,170.435,51.066,159.980
C06723=1016.978,324.924,-145.118,170.429,51.070,159.980
C06724=1016.971,324.676,-145.083,170.422,51.075,159.980
C06725=1016.964,324.428,-145.050,170.416,51.079,159.980
C06726=1016.957,324.181,-145.016,170.409,51.083,159.979
C06727=1016.950,323.934,-144.982,170.402,51.087,159.979
C06728=1016.944,323.686,-144.948,170.396,51.090,159.979
C06729=1016.937,323.438,-144.914,170.389,51.095,159.979
C06730=1016.930,323.191,-144.881,170.383,51.098,159.978
C06731=1016.922,322.921,-144.844,170.375,51.103,159.978
C06732=1016.915,322.653,-144.807,170.369,51.107,159.978
C06733=1016.908,322.384,-144.771,170.361,51.112,159.978
C06734=1016.901,322.115,-144.735,170.355,51.116,159.978
C06735=1016.894,321.867,-144.701,170.347,51.120,159.977
C06736=1016.887,321.619,-144.667,170.341,51.124,159.977
C06737=1016.880,321.372,-144.633,170.334,51.128,159.977
C06738=1016.874,321.124,-144.600,170.328,51.132,159.977
C06739=1016.867,320.877,-144.567,170.322,51.137,159.977
C06740=1016.861,320.629,-144.532,170.315,51.141,159.976
C06741=1016.854,320.381,-144.499,170.309,51.145,159.976
C06742=1016.847,320.134,-144.466,170.302,51.150,159.976
C06743=1016.840,319.886,-144.432,170.296,51.153,159.976
C06744=1016.834,319.638,-144.398,170.289,51.157,159.975
C06745=1016.827,319.391,-144.365,170.283,51.162,159.975
C06746=1016.821,319.143,-144.332,170.276,51.166,159.975
C06747=1016.814,318.895,-144.298,170.271,51.170,159.975
C06748=1016.807,318.648,-144.265,170.263,51.174,159.975
C06749=1016.801,318.400,-144.231,170.257,51.178,159.975
C06750=1016.794,318.153,-144.197,170.251,51.183,159.975
C06751=1016.788,317.905,-144.165,170.244,51.187,159.974
C06752=1016.781,317.657,-144.131,170.238,51.191,159.974
C06753=1016.775,317.410,-144.097,170.232,51.195,159.974
C06754=1016.768,317.161,-144.064,170.225,51.200,159.974
C06755=1016.762,316.914,-144.031,170.219,51.204,159.974
C06756=1016.755,316.667,-143.998,170.212,51.209,159.974
C06757=1016.748,316.419,-143.964,170.206,51.212,159.973
C06758=1016.743,316.171,-143.931,170.200,51.217,159.973
C06759=1016.736,315.924,-143.898,170.193,51.222,159.973
C06760=1016.729,315.676,-143.864,170.187,51.226,159.973
C06761=1016.723,315.428,-143.832,170.181,51.230,159.973
C06762=1016.717,315.181,-143.799,170.174,51.234,159.973
C06763=1016.711,314.933,-143.766,170.168,51.239,159.973
C06764=1016.704,314.685,-143.732,170.163,51.243,159.973
C06765=1016.698,314.437,-143.699,170.156,51.247,159.973
C06766=1016.691,314.190,-143.666,170.150,51.252,159.972
C06767=1016.685,313.942,-143.634,170.144,51.256,159.972
C06768=1016.678,313.694,-143.599,170.138,51.261,159.972
C06769=1016.672,313.447,-143.566,170.131,51.265,159.972
C06770=1016.666,313.199,-143.534,170.125,51.269,159.972
C06771=1016.660,312.952,-143.501,170.119,51.274,159.972
C06772=1016.653,312.704,-143.468,170.112,51.279,159.972
C06773=1016.647,312.455,-143.434,170.107,51.283,159.972
C06774=1016.641,312.208,-143.402,170.100,51.287,159.972
C06775=1016.634,311.961,-143.368,170.094,51.292,159.972
C06776=1016.628,311.713,-143.336,170.088,51.296,159.972
C06777=1016.622,311.466,-143.303,170.082,51.301,159.972
C06778=1016.616,311.218,-143.269,170.076,51.305,159.972
C06779=1016.610,310.970,-143.237,170.069,51.310,159.972
C06780=1016.604,310.723,-143.204,170.064,51.315,159.971
C06781=1016.597,310.475,-143.171,170.057,51.318,159.971
C06782=1016.591,310.227,-143.138,170.051,51.323,159.971
C06783=1016.585,309.979,-143.105,170.045,51.328,159.971
C06784=1016.579,309.731,-143.073,170.039,51.332,159.971
C06785=1016.573,309.484,-143.040,170.033,51.337,159.971
C06786=1016.566,309.236,-143.008,170.027,51.342,159.971
C06787=1016.559,308.988,-142.975,170.021,51.347,159.971
C06788=1016.553,308.740,-142.943,170.014,51.352,159.971
C06789=1016.546,308.493,-142.911,170.008,51.356,159.971
C06790=1016.540,308.244,-142.879,170.003,51.361,159.971
C06791=1016.533,307.981,-142.845,169.996,51.366,159.971
C06792=1016.527,307.718,-142.810,169.990,51.372,159.971
C06793=1016.519,307.454,-142.776,169.983,51.376,159.971
C06794=1016.512,307.190,-142.743,169.977,51.382,159.971
C06795=1016.506,306.942,-142.710,169.971,51.386,159.971
C06796=1016.500,306.695,-142.678,169.964,51.391,159.971
C06797=1016.493,306.447,-142.646,169.959,51.396,159.971
C06798=1016.487,306.199,-142.614,169.952,51.401,159.971
C06799=1016.480,305.951,-142.582,169.946,51.406,159.971
C06800=1016.474,305.703,-142.550,169.941,51.411,159.971
C06801=1016.467,305.456,-142.518,169.934,51.416,159.971
C06802=1016.462,305.208,-142.486,169.928,51.421,159.972
C06803=1016.455,304.960,-142.455,169.922,51.426,159.971
C06804=1016.449,304.713,-142.422,169.916,51.431,159.972
C06805=1016.443,304.465,-142.390,169.910,51.435,159.972
C06806=1016.436,304.217,-142.359,169.904,51.441,159.972
C06807=1016.430,303.968,-142.327,169.898,51.445,159.972
C06808=1016.423,303.721,-142.294,169.893,51.451,159.972
C06809=1016.417,303.473,-142.262,169.886,51.455,159.972
C06810=1016.410,303.225,-142.231,169.881,51.461,159.972
C06811=1016.405,302.978,-142.199,169.874,51.466,159.972
C06812=1016.398,302.730,-142.168,169.869,51.471,159.972
C06813=1016.392,302.482,-142.135,169.863,51.476,159.972
C06814=1016.385,302.234,-142.104,169.856,51.481,159.972
C06815=1016.379,301.986,-142.072,169.851,51.486,159.972
C06816=1016.374,301.738,-142.040,169.845,51.491,159.972
C06817=1016.367,301.491,-142.009,169.839,51.496,159.972
C06818=1016.361,301.242,-141.977,169.833,51.501,159.973
C06819=1016.354,300.994,-141.945,169.827,51.507,159.973
C06820=1016.349,300.747,-141.914,169.822,51.512,159.973
C06821=1016.342,300.499,-141.882,169.816,51.516,159.973
C06822=1016.336,300.251,-141.850,169.810,51.522,159.973
C06823=1016.329,300.003,-141.819,169.804,51.527,159.973
C06824=1016.324,299.755,-141.787,169.799,51.532,159.973
C06825=1016.317,299.507,-141.756,169.792,51.537,159.973
C06826=1016.311,299.259,-141.724,169.787,51.542,159.973
C06827=1016.306,299.012,-141.692,169.780,51.548,159.973
C06828=1016.299,298.764,-141.660,169.775,51.553,159.974
C06829=1016.293,298.516,-141.628,169.769,51.558,159.974
C06830=1016.287,298.268,-141.597,169.763,51.563,159.974
C06831=1016.281,298.020,-141.566,169.757,51.568,159.974
C06832=1016.275,297.772,-141.535,169.752,51.573,159.974
C06833=1016.269,297.524,-141.503,169.746,51.579,159.974
C06834=1016.262,297.276,-141.471,169.740,51.584,159.974
C06835=1016.257,297.029,-141.440,169.735,51.589,159.975
C06836=1016.251,296.780,-141.409,169.728,51.595,159.975
C06837=1016.245,296.533,-141.377,169.723,51.600,159.975
C06838=1016.239,296.285,-141.346,169.718,51.605,159.975
C06839=1016.233,296.037,-141.314,169.711,51.611,159.975
C06840=1016.227,295.788,-141.283,169.706,51.616,159.975
C06841=1016.221,295.541,-141.252,169.700,51.621,159.975
C06842=1016.215,295.293,-141.220,169.694,51.627,159.976
C06843=1016.209,295.045,-141.189,169.689,51.632,159.976
C06844=1016.204,294.797,-141.158,169.682,51.637,159.976
C06845=1016.197,294.549,-141.126,169.677,51.642,159.976
C06846=1016.192,294.301,-141.095,169.672,51.648,159.976
C06847=1016.185,294.054,-141.063,169.665,51.653,159.976
C06848=1016.180,293.808,-141.033,169.660,51.658,159.977
C06849=1016.174,293.561,-141.002,169.655,51.664,159.977
C06850=1016.168,293.314,-140.971,169.648,51.669,159.977
C06851=1016.162,293.067,-140.940,169.643,51.675,159.977
C06852=1016.156,292.820,-140.909,169.638,51.680,159.977
C06853=1016.150,292.573,-140.878,169.632,51.686,159.978
C06854=1016.144,292.326,-140.847,169.626,51.691,159.978
C06855=1016.138,292.079,-140.816,169.621,51.697,159.978
C06856=1016.132,291.831,-140.786,169.615,51.702,159.978
C06857=1016.126,291.583,-140.755,169.610,51.708,159.978
C06858=1016.121,291.335,-140.723,169.604,51.714,159.979
C06859=1016.114,291.087,-140.693,169.598,51.719,159.979
C06860=1016.108,290.839,-140.662,169.593,51.724,159.979
C06861=1016.102,290.591,-140.632,169.587,51.730,159.979
C06862=1016.096,290.343,-140.600,169.582,51.736,159.980
C06863=1016.090,290.095,-140.570,169.576,51.742,159.980
C06864=1016.084,289.847,-140.539,169.570,51.747,159.980
C06865=1016.078,289.599,-140.509,169.564,51.753,159.980
C06866=1016.072,289.351,-140.479,169.559,51.759,159.981
C06867=1016.065,289.103,-140.448,169.553,51.765,159.981
C06868=1016.060,288.855,-140.418,169.548,51.771,159.981
C06869=1016.054,288.607,-140.387,169.542,51.776,159.981
C06870=1016.047,288.358,-140.357,169.537,51.782,159.982
C06871=1016.042,288.111,-140.326,169.531,51.787,159.982
C06872=1016.036,287.862,-140.295,169.525,51.794,159.982
C06873=1016.031,287.615,-140.265,169.520,51.799,159.983
C06874=1016.024,287.366,-140.234,169.514,51.805,159.983
C06875=1016.018,287.118,-140.204,169.509,51.811,159.983
C06876=1016.013,286.870,-140.173,169.503,51.816,159.983
C06877=1016.006,286.622,-140.143,169.498,51.822,159.984
C06878=1016.000,286.374,-140.112,169.492,51.829,159.984
C06879=1015.994,286.127,-140.083,169.487,51.834,159.984
C06880=1015.988,285.879,-140.052,169.481,51.840,159.984
C06881=1015.982,285.631,-140.022,169.476,51.846,159.985
C06882=1015.976,285.382,-139.992,169.470,51.852,159.985
C06883=1015.970,285.134,-139.962,169.465,51.858,159.985
C06884=1015.964,284.886,-139.931,169.460,51.864,159.986
C06885=1015.959,284.638,-139.901,169.454,51.870,159.986
C06886=1015.953,284.390,-139.871,169.449,51.875,159.986
C06887=1015.947,284.141,-139.841,169.443,51.882,159.987
C06888=1015.941,283.894,-139.810,169.438,51.888,159.987
C06889=1015.935,283.645,-139.781,169.432,51.894,159.987
C06890=1015.929,283.398,-139.751,169.426,51.900,159.988
C06891=1015.923,283.150,-139.720,169.421,51.906,159.988
C06892=1015.917,282.901,-139.691,169.415,51.912,159.988
C06893=1015.910,282.653,-139.661,169.410,51.918,159.989
C06894=1015.905,282.405,-139.631,169.404,51.924,159.989
C06895=1015.899,282.157,-139.601,169.399,51.930,159.989
C06896=1015.893,281.908,-139.571,169.393,51.937,159.990
C06897=1015.887,281.661,-139.541,169.388,51.943,159.990
C06898=1015.881,281.412,-139.512,169.382,51.949,159.990
C06899=1015.876,281.165,-139.481,169.378,51.955,159.991
C06900=1015.869,280.917,-139.452,169.372,51.961,159.991
C06901=1015.864,280.669,-139.422,169.367,51.968,159.992
C06902=1015.858,280.420,-139.392,169.361,51.974,159.992
C06903=1015.852,280.172,-139.362,169.356,51.980,159.992
C06904=1015.845,279.924,-139.333,169.350,51.986,159.993
C06905=1015.840,279.675,-139.303,169.345,51.992,159.993
C06906=1015.834,279.427,-139.273,169.340,51.998,159.993
C06907=1015.829,279.187,-139.244,169.335,52.004,159.994
C06908=1015.823,278.946,-139.216,169.329,52.010,159.994
C06909=1015.818,278.706,-139.186,169.324,52.017,159.995
C06910=1015.812,278.464,-139.157,169.319,52.023,159.995
C06911=1015.806,278.224,-139.129,169.313,52.029,159.995
C06912=1015.801,277.984,-139.100,169.308,52.035,159.996
C06913=1015.795,277.743,-139.071,169.304,52.041,159.996
C06914=1015.790,277.502,-139.043,169.299,52.047,159.996
C06915=1015.784,277.254,-139.014,169.293,52.053,159.997
C06916=1015.778,277.006,-138.983,169.287,52.060,159.997
C06917=1015.772,276.758,-138.954,169.282,52.066,159.998
C06918=1015.766,276.510,-138.925,169.276,52.072,159.998
C06919=1015.761,276.261,-138.895,169.272,52.079,159.999
C06920=1015.755,276.013,-138.865,169.266,52.085,159.999
C06921=1015.749,275.765,-138.836,169.261,52.092,159.999
C06922=1015.743,275.517,-138.806,169.256,52.098,160.000
C06923=1015.737,275.269,-138.777,169.250,52.105,160.000
C06924=1015.732,275.021,-138.748,169.245,52.111,160.001
C06925=1015.726,274.773,-138.719,169.240,52.118,160.001
C06926=1015.720,274.524,-138.689,169.235,52.124,160.002
C06927=1015.714,274.276,-138.660,169.229,52.131,160.002
C06928=1015.708,274.028,-138.631,169.223,52.137,160.002
C06929=1015.702,273.779,-138.602,169.219,52.144,160.003
C06930=1015.696,273.531,-138.573,169.213,52.151,160.004
C06931=1015.691,273.282,-138.543,169.209,52.157,160.004
C06932=1015.685,273.035,-138.515,169.203,52.164,160.004
C06933=1015.679,272.787,-138.485,169.197,52.170,160.005
C06934=1015.673,272.538,-138.456,169.193,52.177,160.005
C06935=1015.668,272.290,-138.426,169.187,52.184,160.006
C06936=1015.661,272.042,-138.397,169.181,52.190,160.006
C06937=1015.657,271.794,-138.369,169.177,52.197,160.007
C06938=1015.651,271.545,-138.340,169.171,52.203,160.007
C06939=1015.644,271.297,-138.311,169.166,52.210,160.008
C06940=1015.639,271.049,-138.281,169.161,52.216,160.008
C06941=1015.633,270.801,-138.252,169.156,52.223,160.009
C06942=1015.627,270.553,-138.224,169.151,52.230,160.009
C06943=1015.622,270.304,-138.194,169.146,52.237,160.010
C06944=1015.615,270.056,-138.165,169.140,52.244,160.010
C06945=1015.611,269.808,-138.137,169.135,52.250,160.011
C06946=1015.605,269.560,-138.108,169.130,52.257,160.011
C06947=1015.598,269.311,-138.079,169.124,52.264,160.012
C06948=1015.594,269.063,-138.050,169.120,52.271,160.012
C06949=1015.588,268.815,-138.021,169.114,52.278,160.013
C06950=1015.582,268.566,-137.993,169.109,52.285,160.013
C06951=1015.576,268.319,-137.964,169.104,52.291,160.014
C06952=1015.570,268.070,-137.934,169.099,52.298,160.014
C06953=1015.564,267.822,-137.906,169.094,52.305,160.015
C06954=1015.559,267.574,-137.877,169.088,52.312,160.015
C06955=1015.553,267.325,-137.849,169.084,52.319,160.016
C06956=1015.548,267.076,-137.820,169.078,52.326,160.016
C06957=1015.542,266.829,-137.792,169.073,52.333,160.017
C06958=1015.536,266.580,-137.763,169.068,52.340,160.018
C06959=1015.530,266.332,-137.734,169.063,52.347,160.018
C06960=1015.524,266.084,-137.706,169.057,52.354,160.019
C06961=1015.519,265.836,-137.677,169.052,52.361,160.019
C06962=1015.514,265.587,-137.649,169.047,52.367,160.020
C06963=1015.508,265.339,-137.620,169.042,52.374,160.020
C06964=1015.501,265.091,-137.591,169.037,52.382,160.021
C06965=1015.496,264.843,-137.563,169.031,52.389,160.021
C06966=1015.490,264.594,-137.535,169.027,52.396,160.022
C06967=1015.485,264.355,-137.507,169.022,52.403,160.023
C06968=1015.479,264.117,-137.480,169.017,52.409,160.023
C06969=1015.474,263.878,-137.453,169.012,52.416,160.024
C06970=1015.468,263.640,-137.426,169.007,52.423,160.024
C06971=1015.463,263.402,-137.399,169.002,52.430,160.025
C06972=1015.458,263.163,-137.371,168.997,52.437,160.025
C06973=1015.452,262.925,-137.344,168.992,52.444,160.026
C06974=1015.447,262.686,-137.317,168.987,52.450,160.026
C06975=1015.441,262.438,-137.289,168.982,52.458,160.027
C06976=1015.435,262.190,-137.260,168.977,52.465,160.028
C06977=1015.430,261.941,-137.232,168.973,52.472,160.028
C06978=1015.424,261.693,-137.204,168.968,52.479,160.029
C06979=1015.419,261.445,-137.176,168.962,52.486,160.030
C06980=1015.413,261.196,-137.147,168.957,52.494,160.030
C06981=1015.407,260.948,-137.119,168.952,52.501,160.031
C06982=1015.402,260.700,-137.092,168.947,52.508,160.031
C06983=1015.396,260.451,-137.063,168.942,52.516,160.032
C06984=1015.391,260.203,-137.035,168.937,52.523,160.033
C06985=1015.385,259.954,-137.007,168.932,52.530,160.033
C06986=1015.379,259.706,-136.979,168.926,52.537,160.034
C06987=1015.373,259.457,-136.951,168.921,52.545,160.034
C06988=1015.368,259.209,-136.923,168.916,52.553,160.035
C06989=1015.362,258.962,-136.895,168.912,52.560,160.036
C06990=1015.356,258.713,-136.867,168.907,52.567,160.037
C06991=1015.350,258.465,-136.840,168.902,52.575,160.037
C06992=1015.345,258.217,-136.812,168.897,52.583,160.038
C06993=1015.339,257.968,-136.784,168.892,52.590,160.038
C06994=1015.333,257.720,-136.757,168.887,52.598,160.039
C06995=1015.327,257.471,-136.729,168.882,52.605,160.040
C06996=1015.321,257.223,-136.702,168.877,52.613,160.041
C06997=1015.316,256.975,-136.674,168.871,52.620,160.041
C06998=1015.310,256.725,-136.646,168.866,52.628,160.042
C06999=1015.304,256.478,-136.619,168.861,52.636,160.043
C07000=1015.298,256.228,-136.591,168.856,52.643,160.043
C07001=1015.292,255.981,-136.564,168.851,52.651,160.044
C07002=1015.287,255.733,-136.536,168.846,52.659,160.045
C07003=1015.281,255.483,-136.508,168.841,52.667,160.045
C07004=1015.275,255.235,-136.481,168.836,52.674,160.046
C07005=1015.270,254.987,-136.454,168.831,52.681,160.047
C07006=1015.264,254.738,-136.425,168.826,52.689,160.047
C07007=1015.258,254.490,-136.398,168.821,52.697,160.048
C07008=1015.253,254.242,-136.371,168.816,52.705,160.049
C07009=1015.247,253.994,-136.343,168.811,52.712,160.050
C07010=1015.242,253.745,-136.316,168.806,52.720,160.050
C07011=1015.236,253.496,-136.288,168.801,52.728,160.051
C07012=1015.230,253.248,-136.261,168.796,52.736,160.052
C07013=1015.225,252.999,-136.234,168.791,52.743,160.052
C07014=1015.219,252.751,-136.206,168.786,52.751,160.053
C07015=1015.214,252.502,-136.179,168.781,52.759,160.054
C07016=1015.208,252.254,-136.151,168.776,52.767,160.055
C07017=1015.203,252.006,-136.124,168.771,52.774,160.055
C07018=1015.197,251.757,-136.096,168.766,52.782,160.056
C07019=1015.191,251.509,-136.069,168.761,52.790,160.057
C07020=1015.186,251.260,-136.042,168.757,52.798,160.058
C07021=1015.180,251.012,-136.014,168.752,52.806,160.058
C07022=1015.175,250.764,-135.987,168.747,52.814,160.059
C07023=1015.169,250.514,-135.960,168.742,52.822,160.060
C07024=1015.163,250.267,-135.932,168.737,52.830,160.061
C07025=1015.158,250.018,-135.905,168.732,52.837,160.061
C07026=1015.153,249.769,-135.878,168.727,52.845,160.062
C07027=1015.147,249.531,-135.851,168.722,52.853,160.063
C07028=1015.142,249.291,-135.826,168.718,52.860,160.064
C07029=1015.137,249.051,-135.799,168.713,52.868,160.064
C07030=1015.131,248.812,-135.773,168.708,52.876,160.065
C07031=1015.126,248.572,-135.747,168.705,52.883,160.066
C07032=1015.120,248.334,-135.720,168.700,52.891,160.067
C07033=1015.116,248.094,-135.694,168.695,52.899,160.067
C07034=1015.110,247.855,-135.668,168.690,52.907,160.068
C07035=1015.105,247.606,-135.641,168.685,52.915,160.069
C07036=1015.099,247.357,-135.614,168.680,52.923,160.070
C07037=1015.094,247.108,-135.587,168.675,52.931,160.070
C07038=1015.088,246.861,-135.559,168.671,52.939,160.071
C07039=1015.083,246.612,-135.532,168.666,52.947,160.072
C07040=1015.078,246.363,-135.505,168.661,52.955,160.073
C07041=1015.072,246.115,-135.478,168.657,52.963,160.074
C07042=1015.067,245.866,-135.451,168.652,52.971,160.074
C07043=1015.061,245.618,-135.424,168.647,52.979,160.075
C07044=1015.056,245.369,-135.397,168.642,52.987,160.076
C07045=1015.051,245.121,-135.370,168.636,52.996,160.077
C07046=1015.045,244.872,-135.343,168.632,53.004,160.078
C07047=1015.040,244.624,-135.316,168.627,53.012,160.078
C07048=1015.034,244.376,-135.288,168.622,53.020,160.079
C07049=1015.029,244.127,-135.261,168.617,53.028,160.080
C07050=1015.023,243.879,-135.235,168.613,53.037,160.081
C07051=1015.018,243.630,-135.207,168.608,53.045,160.082
C07052=1015.014,243.382,-135.180,168.604,53.053,160.083
C07053=1015.008,243.134,-135.154,168.599,53.061,160.083
C07054=1015.003,242.885,-135.127,168.594,53.069,160.084
C07055=1014.997,242.637,-135.100,168.588,53.078,160.085
C07056=1014.993,242.388,-135.073,168.584,53.086,160.086
C07057=1014.987,242.139,-135.047,168.579,53.095,160.087
C07058=1014.981,241.891,-135.020,168.574,53.102,160.087
C07059=1014.975,241.642,-134.993,168.570,53.111,160.088
C07060=1014.970,241.394,-134.966,168.565,53.120,160.089
C07061=1014.965,241.145,-134.940,168.560,53.128,160.090
C07062=1014.960,240.897,-134.914,168.555,53.136,160.091
C07063=1014.955,240.648,-134.887,168.551,53.145,160.092
C07064=1014.949,240.400,-134.860,168.545,53.154,160.093
C07065=1014.943,240.151,-134.834,168.541,53.162,160.094
C07066=1014.938,239.903,-134.807,168.536,53.170,160.094
C07067=1014.933,239.654,-134.780,168.532,53.179,160.095
C07068=1014.927,239.405,-134.754,168.526,53.187,160.096
C07069=1014.922,239.157,-134.728,168.522,53.196,160.097
C07070=1014.917,238.909,-134.701,168.517,53.204,160.098
C07071=1014.911,238.660,-134.675,168.513,53.213,160.099
C07072=1014.906,238.411,-134.648,168.507,53.222,160.100
C07073=1014.900,238.163,-134.622,168.503,53.230,160.101
C07074=1014.895,237.915,-134.596,168.498,53.239,160.102
C07075=1014.889,237.666,-134.569,168.493,53.248,160.102
C07076=1014.884,237.417,-134.543,168.489,53.256,160.103
C07077=1014.878,237.169,-134.517,168.484,53.265,160.104
C07078=1014.873,236.920,-134.491,168.479,53.274,160.105
C07079=1014.868,236.672,-134.465,168.474,53.282,160.106
C07080=1014.862,236.424,-134.439,168.470,53.291,160.107
C07081=1014.856,236.175,-134.413,168.464,53.300,160.108
C07082=1014.851,235.926,-134.386,168.460,53.309,160.109
C07083=1014.845,235.677,-134.360,168.455,53.317,160.110
C07084=1014.840,235.429,-134.335,168.451,53.327,160.111
C07085=1014.835,235.181,-134.308,168.446,53.335,160.112
C07086=1014.829,234.932,-134.282,168.441,53.344,160.113
C07087=1014.824,234.689,-134.256,168.436,53.353,160.114
C07088=1014.819,234.446,-134.231,168.432,53.361,160.115
C07089=1014.814,234.203,-134.206,168.428,53.370,160.116
C07090=1014.808,233.960,-134.180,168.422,53.379,160.116
C07091=1014.803,233.718,-134.155,168.418,53.387,160.117
C07092=1014.797,233.475,-134.129,168.413,53.396,160.118
C07093=1014.792,233.232,-134.104,168.409,53.405,160.119
C07094=1014.787,232.989,-134.079,168.404,53.414,160.120
C07095=1014.782,232.741,-134.053,168.400,53.423,160.121
C07096=1014.776,232.492,-134.027,168.395,53.431,160.122
C07097=1014.771,232.243,-134.001,168.390,53.441,160.123
C07098=1014.766,231.994,-133.975,168.386,53.450,160.124
C07099=1014.760,231.745,-133.949,168.380,53.459,160.125
C07100=1014.755,231.498,-133.923,168.377,53.468,160.126
C07101=1014.750,231.249,-133.897,168.371,53.477,160.127
C07102=1014.745,231.001,-133.871,168.367,53.485,160.128
C07103=1014.739,230.752,-133.845,168.362,53.495,160.129
C07104=1014.733,230.503,-133.820,168.357,53.504,160.130
C07105=1014.728,230.255,-133.795,168.352,53.513,160.131
C07106=1014.723,230.006,-133.769,168.348,53.522,160.132
C07107=1014.717,229.757,-133.743,168.343,53.532,160.133
C07108=1014.712,229.509,-133.716,168.339,53.540,160.134
C07109=1014.707,229.260,-133.690,168.334,53.550,160.135
C07110=1014.702,229.012,-133.665,168.330,53.558,160.136
C07111=1014.696,228.763,-133.639,168.325,53.568,160.137
C07112=1014.691,228.515,-133.614,168.320,53.577,160.138
C07113=1014.686,228.265,-133.589,168.315,53.586,160.139
C07114=1014.681,228.017,-133.563,168.311,53.595,160.140
C07115=1014.675,227.768,-133.537,168.306,53.605,160.141
C07116=1014.670,227.519,-133.511,168.301,53.614,160.142
C07117=1014.664,227.271,-133.486,168.297,53.623,160.143
C07118=1014.659,227.022,-133.460,168.292,53.633,160.144
C07119=1014.654,226.774,-133.435,168.288,53.642,160.145
C07120=1014.648,226.525,-133.409,168.283,53.651,160.146
C07121=1014.643,226.277,-133.384,168.278,53.661,160.147
C07122=1014.638,226.027,-133.359,168.274,53.670,160.148
C07123=1014.633,225.779,-133.333,168.269,53.680,160.149
C07124=1014.626,225.530,-133.308,168.264,53.689,160.150
C07125=1014.622,225.282,-133.282,168.260,53.698,160.151
C07126=1014.616,225.033,-133.258,168.255,53.708,160.152
C07127=1014.611,224.784,-133.232,168.250,53.717,160.154
C07128=1014.605,224.536,-133.207,168.246,53.727,160.155
C07129=1014.600,224.287,-133.182,168.241,53.736,160.156
C07130=1014.594,224.038,-133.157,168.236,53.746,160.157
C07131=1014.589,223.790,-133.131,168.232,53.756,160.158
C07132=1014.584,223.541,-133.106,168.228,53.765,160.159
C07133=1014.578,223.292,-133.081,168.223,53.775,160.160
C07134=1014.574,223.043,-133.056,168.218,53.785,160.161
C07135=1014.567,222.795,-133.031,168.214,53.794,160.162
C07136=1014.563,222.546,-133.005,168.209,53.804,160.164
C07137=1014.557,222.297,-132.980,168.204,53.813,160.165
C07138=1014.552,222.049,-132.955,168.199,53.823,160.166
C07139=1014.547,221.800,-132.931,168.196,53.833,160.167
